DATA_BLOCK DB 5001
VERSION : 0.1
  STRUCT
   MODE_NUM : ARRAY  [0 .. 200 ] OF INT  := 0;
   MODE_LIST_TVS : ARRAY  [1000 .. 1009 ] OF STRUCT
    DINT0 : DINT ;
    DINT1 : DINT ;
    DINT2 : DINT ;
   END_STRUCT ;
   MODE_LIST_TVS1 : ARRAY  [1050 .. 1055 ] OF STRUCT
    DINT0 : DINT ;
    DINT1 : DINT ;
    DINT2 : DINT ;
   END_STRUCT ;
   MODE_LIST_TVS2 : ARRAY  [1130 .. 1135 ] OF STRUCT
    DINT0 : DINT ;
    DINT1 : DINT ;
    DINT2 : DINT ;
   END_STRUCT ;
   MODE_LIST_TVS3 : ARRAY  [1150 .. 1155 ] OF STRUCT
    DINT0 : DINT ;
    DINT1 : DINT ;
    DINT2 : DINT ;
   END_STRUCT ;
   MODE_LIST_TVS4 : ARRAY  [1230 .. 1235 ] OF STRUCT
    DINT0 : DINT ;
    DINT1 : DINT ;
    DINT2 : DINT ;
   END_STRUCT ;
   MODE_LIST_TVS5 : ARRAY  [1250 .. 1255 ] OF STRUCT
    DINT0 : DINT ;
    DINT1 : DINT ;
    DINT2 : DINT ;
   END_STRUCT ;
   MODE_LIST_PVS1 : ARRAY  [2000 .. 2015 ] OF STRUCT
    DINT0 : DINT ;
    DINT1 : DINT ;
    DINT2 : DINT ;
   END_STRUCT ;
   MODE_LIST_PVS2 : ARRAY  [2020 .. 2025 ] OF STRUCT
    DINT0 : DINT ;
    DINT1 : DINT ;
    DINT2 : DINT ;
   END_STRUCT ;
   MODE_LIST_PVS3 : ARRAY  [2050 .. 2065 ] OF STRUCT
    DINT0 : DINT ;
    DINT1 : DINT ;
    DINT2 : DINT ;
   END_STRUCT ;
   MODE_LIST_RVS1 : ARRAY  [3000 .. 3015 ] OF STRUCT
    DINT0 : DINT ;
    DINT1 : DINT ;
    DINT2 : DINT ;
    DINT3 : DINT ;
    DINT4 : DINT ;
    DINT5 : DINT ;
    DINT6 : DINT ;
    DINT7 : DINT ;
    DINT8 : DINT ;
    DINT9 : DINT ;
    DINT10 : DINT ;
   END_STRUCT ;
   MODE_LIST_RVS2 : ARRAY  [3020 .. 3040 ] OF STRUCT
    DINT0 : DINT ;
    DINT1 : DINT ;
    DINT2 : DINT ;
    DINT3 : DINT ;
    DINT4 : DINT ;
    DINT5 : DINT ;
    DINT6 : DINT ;
    DINT7 : DINT ;
    DINT8 : DINT ;
    DINT9 : DINT ;
    DINT10 : DINT ;
   END_STRUCT ;
   MODE_LIST_RVS3 : ARRAY  [3050 .. 3080 ] OF STRUCT
    DINT0 : DINT ;
    DINT1 : DINT ;
    DINT2 : DINT ;
    DINT3 : DINT ;
    DINT4 : DINT ;
    DINT5 : DINT ;
    DINT6 : DINT ;
    DINT7 : DINT ;
    DINT8 : DINT ;
    DINT9 : DINT ;
    DINT10 : DINT ;
   END_STRUCT ;
   MODE_LIST_BY : ARRAY  [3100 .. 3105 ] OF STRUCT
    DINT0 : DINT ;
   END_STRUCT ;
  END_STRUCT ;	
BEGIN
   MODE_NUM[0] := 1000;
   MODE_NUM[1] := 1001;
   MODE_NUM[2] := 1002;
   MODE_NUM[3] := 1003;
   MODE_NUM[4] := 1004;
   MODE_NUM[5] := 1005;
   MODE_NUM[6] := 1006;
   MODE_NUM[7] := 1007;
   MODE_NUM[8] := 1008;
   MODE_NUM[9] := 1009;
   MODE_NUM[10] := 1050;
   MODE_NUM[11] := 1051;
   MODE_NUM[12] := 1052;
   MODE_NUM[13] := 1053;
   MODE_NUM[14] := 1054;
   MODE_NUM[15] := 1055;
   MODE_NUM[16] := 1130;
   MODE_NUM[17] := 1131;
   MODE_NUM[18] := 1132;
   MODE_NUM[19] := 1133;
   MODE_NUM[20] := 1134;
   MODE_NUM[21] := 1135;
   MODE_NUM[22] := 1150;
   MODE_NUM[23] := 1151;
   MODE_NUM[24] := 1152;
   MODE_NUM[25] := 1153;
   MODE_NUM[26] := 1154;
   MODE_NUM[27] := 1155;
   MODE_NUM[28] := 1230;
   MODE_NUM[29] := 1231;
   MODE_NUM[30] := 1232;
   MODE_NUM[31] := 1233;
   MODE_NUM[32] := 1234;
   MODE_NUM[33] := 1235;
   MODE_NUM[34] := 1250;
   MODE_NUM[35] := 1251;
   MODE_NUM[36] := 1252;
   MODE_NUM[37] := 1253;
   MODE_NUM[38] := 1254;
   MODE_NUM[39] := 1255;
   MODE_NUM[40] := 2000;
   MODE_NUM[41] := 2001;
   MODE_NUM[42] := 2002;
   MODE_NUM[43] := 2003;
   MODE_NUM[44] := 2004;
   MODE_NUM[45] := 2005;
   MODE_NUM[46] := 2006;
   MODE_NUM[47] := 2007;
   MODE_NUM[48] := 2008;
   MODE_NUM[49] := 2009;
   MODE_NUM[50] := 2010;
   MODE_NUM[51] := 2011;
   MODE_NUM[52] := 2012;
   MODE_NUM[53] := 2013;
   MODE_NUM[54] := 2014;
   MODE_NUM[55] := 2015;
   MODE_NUM[56] := 2020;
   MODE_NUM[57] := 2021;
   MODE_NUM[58] := 2022;
   MODE_NUM[59] := 2023;
   MODE_NUM[60] := 2024;
   MODE_NUM[61] := 2025;
   MODE_NUM[62] := 2050;
   MODE_NUM[63] := 2051;
   MODE_NUM[64] := 2052;
   MODE_NUM[65] := 2053;
   MODE_NUM[66] := 2054;
   MODE_NUM[67] := 2055;
   MODE_NUM[68] := 2056;
   MODE_NUM[69] := 2057;
   MODE_NUM[70] := 2058;
   MODE_NUM[71] := 2059;
   MODE_NUM[72] := 2060;
   MODE_NUM[73] := 2061;
   MODE_NUM[74] := 2062;
   MODE_NUM[75] := 2063;
   MODE_NUM[76] := 2064;
   MODE_NUM[77] := 2065;
   MODE_NUM[78] := 3000;
   MODE_NUM[79] := 3001;
   MODE_NUM[80] := 3002;
   MODE_NUM[81] := 3003;
   MODE_NUM[82] := 3004;
   MODE_NUM[83] := 3005;
   MODE_NUM[84] := 3006;
   MODE_NUM[85] := 3007;
   MODE_NUM[86] := 3008;
   MODE_NUM[87] := 3009;
   MODE_NUM[88] := 3010;
   MODE_NUM[89] := 302;
   MODE_NUM[90] := 3012;
   MODE_NUM[91] := 3013;
   MODE_NUM[92] := 3014;
   MODE_NUM[93] := 3015;
   MODE_NUM[94] := 3020;
   MODE_NUM[95] := 3021;
   MODE_NUM[96] := 3022;
   MODE_NUM[97] := 3023;
   MODE_NUM[98] := 3024;
   MODE_NUM[99] := 3025;
   MODE_NUM[100] := 3026;
   MODE_NUM[101] := 3027;
   MODE_NUM[102] := 3028;
   MODE_NUM[103] := 3029;
   MODE_NUM[104] := 3030;
   MODE_NUM[105] := 3031;
   MODE_NUM[106] := 3032;
   MODE_NUM[107] := 3033;
   MODE_NUM[108] := 3034;
   MODE_NUM[109] := 3035;
   MODE_NUM[110] := 3036;
   MODE_NUM[111] := 3037;
   MODE_NUM[112] := 3038;
   MODE_NUM[113] := 3039;
   MODE_NUM[114] := 3040;
   MODE_NUM[115] := 3050;
   MODE_NUM[116] := 3051;
   MODE_NUM[117] := 3052;
   MODE_NUM[118] := 3053;
   MODE_NUM[119] := 3054;
   MODE_NUM[120] := 3055;
   MODE_NUM[121] := 3056;
   MODE_NUM[122] := 3057;
   MODE_NUM[123] := 3058;
   MODE_NUM[124] := 3059;
   MODE_NUM[125] := 3060;
   MODE_NUM[126] := 3061;
   MODE_NUM[127] := 3062;
   MODE_NUM[128] := 3063;
   MODE_NUM[129] := 3064;
   MODE_NUM[130] := 3065;
   MODE_NUM[131] := 3066;
   MODE_NUM[132] := 3067;
   MODE_NUM[133] := 3068;
   MODE_NUM[134] := 3069;
   MODE_NUM[135] := 3070;
   MODE_NUM[136] := 3071;
   MODE_NUM[137] := 3072;
   MODE_NUM[138] := 3073;
   MODE_NUM[139] := 3074;
   MODE_NUM[140] := 3075;
   MODE_NUM[141] := 3076;
   MODE_NUM[142] := 3077;
   MODE_NUM[143] := 3078;
   MODE_NUM[144] := 3079;
   MODE_NUM[145] := 3080;
   MODE_LIST_TVS[1000].DINT0 := L#1475696127;
   MODE_LIST_TVS[1000].DINT1 := L#1431697397;
   MODE_LIST_TVS[1001].DINT0 := L#-580919467;
   MODE_LIST_TVS[1001].DINT1 := L#-8865;
   MODE_LIST_TVS[1002].DINT0 := L#-44171350;
   MODE_LIST_TVS[1002].DINT1 := L#-33443;
   MODE_LIST_TVS[1003].DINT0 := L#-547496107;
   MODE_LIST_TVS[1003].DINT1 := L#1431699293;
   MODE_LIST_TVS[1004].DINT0 := L#-547496022;
   MODE_LIST_TVS[1004].DINT1 := L#1431699293;
   MODE_LIST_TVS[1005].DINT0 := L#1609916415;
   MODE_LIST_TVS[1005].DINT1 := L#1431699445;
   MODE_LIST_TVS1[1050].DINT0 := L#-142779785;
   MODE_LIST_TVS1[1050].DINT1 := L#-572655747;
   MODE_LIST_TVS1[1051].DINT0 := L#-673850659;
   MODE_LIST_TVS1[1051].DINT1 := L#-572655649;
   MODE_LIST_TVS1[1052].DINT0 := L#-142779785;
   MODE_LIST_TVS1[1052].DINT1 := L#-572688513;
   MODE_LIST_TVS1[1053].DINT0 := L#-136979747;
   MODE_LIST_TVS1[1053].DINT1 := L#-572663841;
   MODE_LIST_TVS4[1230].DINT0 := L#1609916351;
   MODE_LIST_TVS4[1230].DINT1 := L#1431699325;
   MODE_LIST_TVS4[1231].DINT0 := L#-537567249;
   MODE_LIST_TVS4[1231].DINT1 := L#1431699413;
   MODE_LIST_TVS4[1232].DINT0 := L#-537567313;
   MODE_LIST_TVS4[1232].DINT1 := L#1431699293;
   MODE_LIST_TVS5[1250].DINT0 := L#-142779817;
   MODE_LIST_TVS5[1250].DINT1 := L#-572656291;
   MODE_LIST_TVS5[1251].DINT0 := L#1602052027;
   MODE_LIST_TVS5[1251].DINT1 := L#1431699325;
   MODE_LIST_TVS5[1252].DINT0 := L#-539631634;
   MODE_LIST_TVS5[1252].DINT1 := L#1431699413;
   MODE_LIST_TVS5[1253].DINT0 := L#-673850787;
   MODE_LIST_TVS5[1253].DINT1 := L#-572656289;
   MODE_LIST_PVS1[2000].DINT0 := L#-356515841;
   MODE_LIST_PVS1[2000].DINT1 := L#-1;
   MODE_LIST_PVS1[2000].DINT2 := L#16383;
   MODE_LIST_PVS1[2001].DINT0 := L#-356518571;
   MODE_LIST_PVS1[2001].DINT1 := L#-305291;
   MODE_LIST_PVS1[2001].DINT2 := L#15735;
   MODE_LIST_PVS1[2002].DINT0 := L#1790965077;
   MODE_LIST_PVS1[2002].DINT1 := L#-41515;
   MODE_LIST_PVS1[2002].DINT2 := L#15829;
   MODE_LIST_PVS1[2003].DINT0 := L#1790965077;
   MODE_LIST_PVS1[2003].DINT1 := L#-41515;
   MODE_LIST_PVS1[2003].DINT2 := L#15829;
   MODE_LIST_PVS1[2004].DINT0 := L#1790965077;
   MODE_LIST_PVS1[2004].DINT1 := L#-41515;
   MODE_LIST_PVS1[2004].DINT2 := L#15829;
   MODE_LIST_PVS1[2005].DINT0 := L#-1;
   MODE_LIST_PVS1[2005].DINT1 := L#-1;
   MODE_LIST_PVS1[2005].DINT2 := L#16383;
   MODE_LIST_PVS1[2006].DINT0 := L#1434449237;
   MODE_LIST_PVS1[2006].DINT1 := L#3888469;
   MODE_LIST_PVS1[2006].DINT2 := L#15701;
   MODE_LIST_PVS1[2007].DINT0 := L#1790967765;
   MODE_LIST_PVS1[2007].DINT1 := L#4194293;
   MODE_LIST_PVS1[2007].DINT2 := L#16373;
   MODE_LIST_PVS1[2008].DINT0 := L#-356518529;
   MODE_LIST_PVS1[2008].DINT1 := L#4152799;
   MODE_LIST_PVS1[2008].DINT2 := L#15839;
   MODE_LIST_PVS1[2009].DINT0 := L#-1;
   MODE_LIST_PVS1[2009].DINT1 := L#-1;
   MODE_LIST_PVS1[2009].DINT2 := L#16383;
   MODE_LIST_PVS1[2010].DINT0 := L#-143261697;
   MODE_LIST_PVS1[2010].DINT1 := L#4059103;
   MODE_LIST_PVS1[2010].DINT2 := L#14335;
   MODE_LIST_PVS1[2011].DINT0 := L#-143261697;
   MODE_LIST_PVS1[2011].DINT1 := L#4059103;
   MODE_LIST_PVS1[2011].DINT2 := L#14335;
   MODE_LIST_PVS3[2050].DINT0 := L#-1019224065;
   MODE_LIST_PVS3[2050].DINT1 := L#3670015;
   MODE_LIST_PVS3[2050].DINT2 := L#16383;
   MODE_LIST_PVS3[2051].DINT0 := L#-600309761;
   MODE_LIST_PVS3[2051].DINT1 := L#4194303;
   MODE_LIST_PVS3[2051].DINT2 := L#14335;
   MODE_LIST_PVS3[2052].DINT0 := L#-1069580289;
   MODE_LIST_PVS3[2052].DINT1 := L#2145386495;
   MODE_LIST_PVS3[2052].DINT2 := L#16383;
   MODE_LIST_PVS3[2053].DINT0 := L#-1069580289;
   MODE_LIST_PVS3[2053].DINT1 := L#-10485761;
   MODE_LIST_PVS3[2053].DINT2 := L#16383;
   MODE_LIST_PVS3[2054].DINT0 := L#-1069580289;
   MODE_LIST_PVS3[2054].DINT1 := L#-673185793;
   MODE_LIST_PVS3[2054].DINT2 := L#16383;
   MODE_LIST_PVS3[2055].DINT0 := L#-1069580289;
   MODE_LIST_PVS3[2055].DINT1 := L#-35651585;
   MODE_LIST_PVS3[2055].DINT2 := L#16383;
   MODE_LIST_PVS3[2056].DINT0 := L#-1071644673;
   MODE_LIST_PVS3[2056].DINT1 := L#4194303;
   MODE_LIST_PVS3[2056].DINT2 := L#8191;
   MODE_LIST_PVS3[2057].DINT0 := L#-143261697;
   MODE_LIST_PVS3[2057].DINT1 := L#4059103;
   MODE_LIST_PVS3[2057].DINT2 := L#14335;
   MODE_LIST_RVS1[3000].DINT0 := L#1431666687;
   MODE_LIST_RVS1[3000].DINT1 := L#-11;
   MODE_LIST_RVS1[3000].DINT2 := L#-1;
   MODE_LIST_RVS1[3000].DINT3 := L#1431656447;
   MODE_LIST_RVS1[3000].DINT4 := L#1431655765;
   MODE_LIST_RVS1[3000].DINT5 := L#-43;
   MODE_LIST_RVS1[3000].DINT6 := L#-1;
   MODE_LIST_RVS1[3000].DINT7 := L#1432354815;
   MODE_LIST_RVS1[3000].DINT8 := L#-43691;
   MODE_LIST_RVS1[3000].DINT9 := L#-1;
   MODE_LIST_RVS1[3000].DINT10 := L#255;
   MODE_LIST_RVS1[3001].DINT0 := L#16383;
   MODE_LIST_RVS1[3001].DINT1 := L#-16;
   MODE_LIST_RVS1[3001].DINT2 := L#-1;
   MODE_LIST_RVS1[3001].DINT3 := L#1023;
   MODE_LIST_RVS1[3001].DINT5 := L#-64;
   MODE_LIST_RVS1[3001].DINT6 := L#-1;
   MODE_LIST_RVS1[3001].DINT7 := L#1048575;
   MODE_LIST_RVS1[3001].DINT8 := L#-65536;
   MODE_LIST_RVS1[3001].DINT9 := L#-1;
   MODE_LIST_RVS1[3001].DINT10 := L#255;
   MODE_LIST_RVS1[3002].DINT0 := L#10069;
   MODE_LIST_RVS1[3002].DINT1 := L#-707406000;
   MODE_LIST_RVS1[3002].DINT2 := L#1507164117;
   MODE_LIST_RVS1[3002].DINT3 := L#629;
   MODE_LIST_RVS1[3002].DINT5 := L#2012599616;
   MODE_LIST_RVS1[3002].DINT6 := L#-170568363;
   MODE_LIST_RVS1[3002].DINT7 := L#644479;
   MODE_LIST_RVS1[3002].DINT8 := L#1567948800;
   MODE_LIST_RVS1[3002].DINT9 := L#1567972725;
   MODE_LIST_RVS1[3002].DINT10 := L#255;
   MODE_LIST_RVS1[3003].DINT0 := L#7509;
   MODE_LIST_RVS1[3003].DINT1 := L#-707406000;
   MODE_LIST_RVS1[3003].DINT2 := L#1465221077;
   MODE_LIST_RVS1[3003].DINT3 := L#469;
   MODE_LIST_RVS1[3003].DINT5 := L#2012599616;
   MODE_LIST_RVS1[3003].DINT6 := L#-170568363;
   MODE_LIST_RVS1[3003].DINT7 := L#480639;
   MODE_LIST_RVS1[3003].DINT8 := L#1567948800;
   MODE_LIST_RVS1[3003].DINT9 := L#1567972725;
   MODE_LIST_RVS1[3003].DINT10 := L#255;
   MODE_LIST_RVS1[3004].DINT0 := L#7509;
   MODE_LIST_RVS1[3004].DINT1 := L#-707406000;
   MODE_LIST_RVS1[3004].DINT2 := L#1465221077;
   MODE_LIST_RVS1[3004].DINT3 := L#469;
   MODE_LIST_RVS1[3004].DINT5 := L#1442174272;
   MODE_LIST_RVS1[3004].DINT6 := L#-170568363;
   MODE_LIST_RVS1[3004].DINT7 := L#480639;
   MODE_LIST_RVS1[3004].DINT8 := L#1567948800;
   MODE_LIST_RVS1[3004].DINT9 := L#1567972725;
   MODE_LIST_RVS1[3004].DINT10 := L#255;
   MODE_LIST_RVS1[3005].DINT0 := L#7509;
   MODE_LIST_RVS1[3005].DINT1 := L#-707406000;
   MODE_LIST_RVS1[3005].DINT2 := L#1507164117;
   MODE_LIST_RVS1[3005].DINT3 := L#469;
   MODE_LIST_RVS1[3005].DINT5 := L#1442174272;
   MODE_LIST_RVS1[3005].DINT6 := L#-170568363;
   MODE_LIST_RVS1[3005].DINT7 := L#480639;
   MODE_LIST_RVS1[3005].DINT8 := L#1567948800;
   MODE_LIST_RVS1[3005].DINT9 := L#1567972725;
   MODE_LIST_RVS1[3005].DINT10 := L#255;
   MODE_LIST_RVS1[3006].DINT0 := L#16383;
   MODE_LIST_RVS1[3006].DINT1 := L#-16;
   MODE_LIST_RVS1[3006].DINT2 := L#-10944;
   MODE_LIST_RVS1[3006].DINT3 := L#1023;
   MODE_LIST_RVS1[3006].DINT5 := L#-8521792;
   MODE_LIST_RVS1[3006].DINT6 := L#2147221504;
   MODE_LIST_RVS1[3006].DINT7 := L#1048533;
   MODE_LIST_RVS1[3006].DINT8 := L#268369920;
   MODE_LIST_RVS1[3006].DINT9 := L#268374015;
   MODE_LIST_RVS1[3006].DINT10 := L#85;
   MODE_LIST_RVS2[3020].DINT0 := L#1431657813;
   MODE_LIST_RVS2[3020].DINT1 := L#-11;
   MODE_LIST_RVS2[3020].DINT2 := L#-64;
   MODE_LIST_RVS2[3020].DINT3 := L#1023;
   MODE_LIST_RVS2[3020].DINT5 := L#-8521792;
   MODE_LIST_RVS2[3020].DINT6 := L#-262144;
   MODE_LIST_RVS2[3020].DINT7 := L#1048575;
   MODE_LIST_RVS2[3020].DINT8 := L#268369920;
   MODE_LIST_RVS2[3020].DINT9 := L#268374015;
   MODE_LIST_RVS2[3020].DINT10 := L#255;
   MODE_LIST_RVS2[3021].DINT0 := L#1431657813;
   MODE_LIST_RVS2[3021].DINT1 := L#-11;
   MODE_LIST_RVS2[3021].DINT2 := L#-64;
   MODE_LIST_RVS2[3021].DINT3 := L#1023;
   MODE_LIST_RVS2[3021].DINT5 := L#-8521792;
   MODE_LIST_RVS2[3021].DINT6 := L#-262144;
   MODE_LIST_RVS2[3021].DINT7 := L#1048575;
   MODE_LIST_RVS2[3021].DINT8 := L#268369920;
   MODE_LIST_RVS2[3021].DINT9 := L#268374015;
   MODE_LIST_RVS2[3021].DINT10 := L#255;
   MODE_LIST_RVS2[3022].DINT0 := L#1431657813;
   MODE_LIST_RVS2[3022].DINT1 := L#-11;
   MODE_LIST_RVS2[3022].DINT2 := L#-64;
   MODE_LIST_RVS2[3022].DINT3 := L#1023;
   MODE_LIST_RVS2[3022].DINT5 := L#-8521792;
   MODE_LIST_RVS2[3022].DINT6 := L#-262144;
   MODE_LIST_RVS2[3022].DINT7 := L#1048575;
   MODE_LIST_RVS2[3022].DINT8 := L#268369920;
   MODE_LIST_RVS2[3022].DINT9 := L#268374015;
   MODE_LIST_RVS2[3022].DINT10 := L#255;
   MODE_LIST_RVS2[3023].DINT0 := L#1431657813;
   MODE_LIST_RVS2[3023].DINT1 := L#-11;
   MODE_LIST_RVS2[3023].DINT2 := L#-64;
   MODE_LIST_RVS2[3023].DINT3 := L#1023;
   MODE_LIST_RVS2[3023].DINT5 := L#-8521792;
   MODE_LIST_RVS2[3023].DINT6 := L#-262144;
   MODE_LIST_RVS2[3023].DINT7 := L#1048575;
   MODE_LIST_RVS2[3023].DINT8 := L#268369920;
   MODE_LIST_RVS2[3023].DINT9 := L#268374015;
   MODE_LIST_RVS2[3023].DINT10 := L#255;
   MODE_LIST_RVS2[3024].DINT0 := L#16383;
   MODE_LIST_RVS2[3024].DINT1 := L#-16;
   MODE_LIST_RVS2[3024].DINT2 := L#1610612672;
   MODE_LIST_RVS2[3024].DINT3 := L#1431655893;
   MODE_LIST_RVS2[3024].DINT4 := L#1431655765;
   MODE_LIST_RVS2[3024].DINT5 := L#-8521771;
   MODE_LIST_RVS2[3024].DINT6 := L#-262144;
   MODE_LIST_RVS2[3024].DINT7 := L#1048575;
   MODE_LIST_RVS2[3024].DINT8 := L#268369920;
   MODE_LIST_RVS2[3024].DINT9 := L#268374015;
   MODE_LIST_RVS2[3024].DINT10 := L#255;
   MODE_LIST_RVS2[3025].DINT0 := L#16383;
   MODE_LIST_RVS2[3025].DINT1 := L#-16;
   MODE_LIST_RVS2[3025].DINT2 := L#1610612672;
   MODE_LIST_RVS2[3025].DINT3 := L#1431655893;
   MODE_LIST_RVS2[3025].DINT4 := L#1431655765;
   MODE_LIST_RVS2[3025].DINT5 := L#-8521771;
   MODE_LIST_RVS2[3025].DINT6 := L#-262144;
   MODE_LIST_RVS2[3025].DINT7 := L#1048575;
   MODE_LIST_RVS2[3025].DINT8 := L#268369920;
   MODE_LIST_RVS2[3025].DINT9 := L#268374015;
   MODE_LIST_RVS2[3025].DINT10 := L#255;
   MODE_LIST_RVS2[3026].DINT0 := L#16383;
   MODE_LIST_RVS2[3026].DINT1 := L#-16;
   MODE_LIST_RVS2[3026].DINT2 := L#1610612672;
   MODE_LIST_RVS2[3026].DINT3 := L#1431655893;
   MODE_LIST_RVS2[3026].DINT4 := L#1431655765;
   MODE_LIST_RVS2[3026].DINT5 := L#-8521771;
   MODE_LIST_RVS2[3026].DINT6 := L#-262144;
   MODE_LIST_RVS2[3026].DINT7 := L#1048575;
   MODE_LIST_RVS2[3026].DINT8 := L#268369920;
   MODE_LIST_RVS2[3026].DINT9 := L#268374015;
   MODE_LIST_RVS2[3026].DINT10 := L#255;
   MODE_LIST_RVS2[3027].DINT0 := L#16383;
   MODE_LIST_RVS2[3027].DINT1 := L#-16;
   MODE_LIST_RVS2[3027].DINT2 := L#1610612672;
   MODE_LIST_RVS2[3027].DINT3 := L#1431655893;
   MODE_LIST_RVS2[3027].DINT4 := L#1431655765;
   MODE_LIST_RVS2[3027].DINT5 := L#-8521771;
   MODE_LIST_RVS2[3027].DINT6 := L#-262144;
   MODE_LIST_RVS2[3027].DINT7 := L#1048575;
   MODE_LIST_RVS2[3027].DINT8 := L#268369920;
   MODE_LIST_RVS2[3027].DINT9 := L#268374015;
   MODE_LIST_RVS2[3027].DINT10 := L#255;
   MODE_LIST_RVS2[3028].DINT0 := L#16383;
   MODE_LIST_RVS2[3028].DINT1 := L#-16;
   MODE_LIST_RVS2[3028].DINT2 := L#1610612672;
   MODE_LIST_RVS2[3028].DINT3 := L#1431655893;
   MODE_LIST_RVS2[3028].DINT4 := L#1431655765;
   MODE_LIST_RVS2[3028].DINT5 := L#-8521771;
   MODE_LIST_RVS2[3028].DINT6 := L#-262144;
   MODE_LIST_RVS2[3028].DINT7 := L#1048575;
   MODE_LIST_RVS2[3028].DINT8 := L#268369920;
   MODE_LIST_RVS2[3028].DINT9 := L#268374015;
   MODE_LIST_RVS2[3028].DINT10 := L#255;
   MODE_LIST_RVS2[3029].DINT0 := L#16383;
   MODE_LIST_RVS2[3029].DINT1 := L#-16;
   MODE_LIST_RVS2[3029].DINT2 := L#1610612672;
   MODE_LIST_RVS2[3029].DINT3 := L#1431655893;
   MODE_LIST_RVS2[3029].DINT4 := L#1431655765;
   MODE_LIST_RVS2[3029].DINT5 := L#-8521771;
   MODE_LIST_RVS2[3029].DINT6 := L#-262144;
   MODE_LIST_RVS2[3029].DINT7 := L#1048575;
   MODE_LIST_RVS2[3029].DINT8 := L#268369920;
   MODE_LIST_RVS2[3029].DINT9 := L#268374015;
   MODE_LIST_RVS2[3029].DINT10 := L#255;
   MODE_LIST_RVS2[3030].DINT0 := L#16383;
   MODE_LIST_RVS2[3030].DINT1 := L#-16;
   MODE_LIST_RVS2[3030].DINT2 := L#1610612672;
   MODE_LIST_RVS2[3030].DINT3 := L#1431655893;
   MODE_LIST_RVS2[3030].DINT4 := L#1431655765;
   MODE_LIST_RVS2[3030].DINT5 := L#-8521771;
   MODE_LIST_RVS2[3030].DINT6 := L#-262144;
   MODE_LIST_RVS2[3030].DINT7 := L#1048575;
   MODE_LIST_RVS2[3030].DINT8 := L#268369920;
   MODE_LIST_RVS2[3030].DINT9 := L#268374015;
   MODE_LIST_RVS2[3030].DINT10 := L#255;
   MODE_LIST_RVS2[3031].DINT0 := L#16383;
   MODE_LIST_RVS2[3031].DINT1 := L#-16;
   MODE_LIST_RVS2[3031].DINT2 := L#1610612672;
   MODE_LIST_RVS2[3031].DINT3 := L#1431655893;
   MODE_LIST_RVS2[3031].DINT4 := L#1431655765;
   MODE_LIST_RVS2[3031].DINT5 := L#-8521771;
   MODE_LIST_RVS2[3031].DINT6 := L#-262144;
   MODE_LIST_RVS2[3031].DINT7 := L#1048575;
   MODE_LIST_RVS2[3031].DINT8 := L#268369920;
   MODE_LIST_RVS2[3031].DINT9 := L#268374015;
   MODE_LIST_RVS2[3031].DINT10 := L#255;
   MODE_LIST_RVS2[3032].DINT0 := L#16383;
   MODE_LIST_RVS2[3032].DINT1 := L#-16;
   MODE_LIST_RVS2[3032].DINT2 := L#1610612672;
   MODE_LIST_RVS2[3032].DINT3 := L#1431655893;
   MODE_LIST_RVS2[3032].DINT4 := L#1431655765;
   MODE_LIST_RVS2[3032].DINT5 := L#-8521771;
   MODE_LIST_RVS2[3032].DINT6 := L#-262144;
   MODE_LIST_RVS2[3032].DINT7 := L#1048575;
   MODE_LIST_RVS2[3032].DINT8 := L#268369920;
   MODE_LIST_RVS2[3032].DINT9 := L#268374015;
   MODE_LIST_RVS2[3032].DINT10 := L#255;
   MODE_LIST_RVS2[3033].DINT0 := L#16383;
   MODE_LIST_RVS2[3033].DINT1 := L#-16;
   MODE_LIST_RVS2[3033].DINT2 := L#1610612672;
   MODE_LIST_RVS2[3033].DINT3 := L#1431655893;
   MODE_LIST_RVS2[3033].DINT4 := L#1431655765;
   MODE_LIST_RVS2[3033].DINT5 := L#-8521771;
   MODE_LIST_RVS2[3033].DINT6 := L#-262144;
   MODE_LIST_RVS2[3033].DINT7 := L#1048575;
   MODE_LIST_RVS2[3033].DINT8 := L#268369920;
   MODE_LIST_RVS2[3033].DINT9 := L#268374015;
   MODE_LIST_RVS2[3033].DINT10 := L#255;
   MODE_LIST_RVS2[3034].DINT0 := L#4178175;
   MODE_LIST_RVS2[3034].DINT2 := L#65280;
   MODE_LIST_RVS2[3034].DINT3 := L#1073725440;
   MODE_LIST_RVS2[3034].DINT5 := L#-8521792;
   MODE_LIST_RVS2[3034].DINT6 := L#-262144;
   MODE_LIST_RVS2[3034].DINT7 := L#-16777153;
   MODE_LIST_RVS2[3034].DINT8 := L#-66060289;
   MODE_LIST_RVS2[3034].DINT9 := L#1073741823;
   MODE_LIST_RVS2[3035].DINT0 := L#16383;
   MODE_LIST_RVS2[3035].DINT1 := L#-16;
   MODE_LIST_RVS2[3035].DINT2 := L#-64;
   MODE_LIST_RVS2[3035].DINT3 := L#1023;
   MODE_LIST_RVS2[3035].DINT5 := L#-8521792;
   MODE_LIST_RVS2[3035].DINT6 := L#-262144;
   MODE_LIST_RVS2[3035].DINT7 := L#1431786879;
   MODE_LIST_RVS2[3035].DINT8 := L#268391765;
   MODE_LIST_RVS2[3035].DINT9 := L#268374015;
   MODE_LIST_RVS2[3035].DINT10 := L#255;
   MODE_LIST_RVS2[3036].DINT0 := L#16383;
   MODE_LIST_RVS2[3036].DINT1 := L#-16;
   MODE_LIST_RVS2[3036].DINT2 := L#-64;
   MODE_LIST_RVS2[3036].DINT3 := L#1023;
   MODE_LIST_RVS2[3036].DINT5 := L#-8521792;
   MODE_LIST_RVS2[3036].DINT6 := L#-262144;
   MODE_LIST_RVS2[3036].DINT7 := L#1431786879;
   MODE_LIST_RVS2[3036].DINT8 := L#268391765;
   MODE_LIST_RVS2[3036].DINT9 := L#268374015;
   MODE_LIST_RVS2[3036].DINT10 := L#255;
   MODE_LIST_RVS2[3037].DINT0 := L#16383;
   MODE_LIST_RVS2[3037].DINT1 := L#-16;
   MODE_LIST_RVS2[3037].DINT2 := L#-64;
   MODE_LIST_RVS2[3037].DINT3 := L#1023;
   MODE_LIST_RVS2[3037].DINT5 := L#-8521792;
   MODE_LIST_RVS2[3037].DINT6 := L#-262144;
   MODE_LIST_RVS2[3037].DINT7 := L#1431786879;
   MODE_LIST_RVS2[3037].DINT8 := L#268391765;
   MODE_LIST_RVS2[3037].DINT9 := L#268374015;
   MODE_LIST_RVS2[3037].DINT10 := L#255;
   MODE_LIST_RVS2[3038].DINT0 := L#16383;
   MODE_LIST_RVS2[3038].DINT1 := L#-16;
   MODE_LIST_RVS2[3038].DINT2 := L#-64;
   MODE_LIST_RVS2[3038].DINT3 := L#1023;
   MODE_LIST_RVS2[3038].DINT5 := L#-8521792;
   MODE_LIST_RVS2[3038].DINT6 := L#-262144;
   MODE_LIST_RVS2[3038].DINT7 := L#1431786879;
   MODE_LIST_RVS2[3038].DINT8 := L#268391765;
   MODE_LIST_RVS2[3038].DINT9 := L#268374015;
   MODE_LIST_RVS2[3038].DINT10 := L#255;
   MODE_LIST_RVS2[3039].DINT0 := L#16383;
   MODE_LIST_RVS2[3039].DINT1 := L#-16;
   MODE_LIST_RVS2[3039].DINT2 := L#-64;
   MODE_LIST_RVS2[3039].DINT3 := L#1023;
   MODE_LIST_RVS2[3039].DINT5 := L#-8521792;
   MODE_LIST_RVS2[3039].DINT6 := L#-262144;
   MODE_LIST_RVS2[3039].DINT7 := L#1431786879;
   MODE_LIST_RVS2[3039].DINT8 := L#268391765;
   MODE_LIST_RVS2[3039].DINT9 := L#268374015;
   MODE_LIST_RVS2[3039].DINT10 := L#255;
   MODE_LIST_RVS3[3050].DINT0 := L#-1;
   MODE_LIST_RVS3[3050].DINT1 := L#255;
   MODE_LIST_RVS3[3050].DINT2 := L#4194048;
   MODE_LIST_RVS3[3050].DINT3 := L#-581091328;
   MODE_LIST_RVS3[3050].DINT4 := L#262133;
   MODE_LIST_RVS3[3050].DINT5 := L#-8521792;
   MODE_LIST_RVS3[3050].DINT6 := L#2147221504;
   MODE_LIST_RVS3[3050].DINT7 := L#1007681493;
   MODE_LIST_RVS3[3050].DINT8 := L#-168296512;
   MODE_LIST_RVS3[3050].DINT9 := L#-43523;
   MODE_LIST_RVS3[3050].DINT10 := L#4095;
   MODE_LIST_RVS3[3051].DINT0 := L#268435455;
   MODE_LIST_RVS3[3051].DINT1 := L#15;
   MODE_LIST_RVS3[3051].DINT2 := L#4194048;
   MODE_LIST_RVS3[3051].DINT3 := L#-581091328;
   MODE_LIST_RVS3[3051].DINT4 := L#262133;
   MODE_LIST_RVS3[3051].DINT5 := L#-8521792;
   MODE_LIST_RVS3[3051].DINT6 := L#2147221504;
   MODE_LIST_RVS3[3051].DINT7 := L#-1070530603;
   MODE_LIST_RVS3[3051].DINT8 := L#-168296512;
   MODE_LIST_RVS3[3051].DINT9 := L#-43523;
   MODE_LIST_RVS3[3051].DINT10 := L#4095;
   MODE_LIST_RVS3[3052].DINT0 := L#12599295;
   MODE_LIST_RVS3[3052].DINT1 := L#-4;
   MODE_LIST_RVS3[3052].DINT2 := L#-10944;
   MODE_LIST_RVS3[3052].DINT3 := L#1023;
   MODE_LIST_RVS3[3052].DINT5 := L#-8521792;
   MODE_LIST_RVS3[3052].DINT6 := L#2147221504;
   MODE_LIST_RVS3[3052].DINT7 := L#1048533;
   MODE_LIST_RVS3[3052].DINT8 := L#268369920;
   MODE_LIST_RVS3[3052].DINT9 := L#268374015;
   MODE_LIST_RVS3[3052].DINT10 := L#85;
   MODE_LIST_RVS3[3053].DINT0 := L#-1070579713;
   MODE_LIST_RVS3[3053].DINT1 := L#-13;
   MODE_LIST_RVS3[3053].DINT2 := L#-10944;
   MODE_LIST_RVS3[3053].DINT3 := L#1023;
   MODE_LIST_RVS3[3053].DINT5 := L#-8521792;
   MODE_LIST_RVS3[3053].DINT6 := L#2147221504;
   MODE_LIST_RVS3[3053].DINT7 := L#1048533;
   MODE_LIST_RVS3[3053].DINT8 := L#268369920;
   MODE_LIST_RVS3[3053].DINT9 := L#268374015;
   MODE_LIST_RVS3[3053].DINT10 := L#85;
   MODE_LIST_RVS3[3054].DINT0 := L#16383;
   MODE_LIST_RVS3[3054].DINT1 := L#-16;
   MODE_LIST_RVS3[3054].DINT2 := L#-10944;
   MODE_LIST_RVS3[3054].DINT3 := L#1023;
   MODE_LIST_RVS3[3054].DINT5 := L#-8521792;
   MODE_LIST_RVS3[3054].DINT6 := L#2147221504;
   MODE_LIST_RVS3[3054].DINT7 := L#1048533;
   MODE_LIST_RVS3[3054].DINT8 := L#268369920;
   MODE_LIST_RVS3[3054].DINT9 := L#268374015;
   MODE_LIST_RVS3[3054].DINT10 := L#85;
   MODE_LIST_RVS3[3055].DINT0 := L#16383;
   MODE_LIST_RVS3[3055].DINT1 := L#-35376;
   MODE_LIST_RVS3[3055].DINT2 := L#-10944;
   MODE_LIST_RVS3[3055].DINT3 := L#1023;
   MODE_LIST_RVS3[3055].DINT5 := L#-8521792;
   MODE_LIST_RVS3[3055].DINT6 := L#2147221504;
   MODE_LIST_RVS3[3055].DINT7 := L#1048533;
   MODE_LIST_RVS3[3055].DINT8 := L#268369920;
   MODE_LIST_RVS3[3055].DINT9 := L#268374015;
   MODE_LIST_RVS3[3055].DINT10 := L#85;
   MODE_LIST_RVS3[3056].DINT0 := L#16383;
   MODE_LIST_RVS3[3056].DINT1 := L#2105409520;
   MODE_LIST_RVS3[3056].DINT2 := L#-10881;
   MODE_LIST_RVS3[3056].DINT3 := L#1023;
   MODE_LIST_RVS3[3056].DINT5 := L#-8521792;
   MODE_LIST_RVS3[3056].DINT6 := L#2147221504;
   MODE_LIST_RVS3[3056].DINT7 := L#1048533;
   MODE_LIST_RVS3[3056].DINT8 := L#268369920;
   MODE_LIST_RVS3[3056].DINT9 := L#268374015;
   MODE_LIST_RVS3[3056].DINT10 := L#85;
   MODE_LIST_RVS3[3057].DINT0 := L#16383;
   MODE_LIST_RVS3[3057].DINT1 := L#-16;
   MODE_LIST_RVS3[3057].DINT2 := L#-10944;
   MODE_LIST_RVS3[3057].DINT3 := L#1023;
   MODE_LIST_RVS3[3057].DINT5 := L#-8521792;
   MODE_LIST_RVS3[3057].DINT6 := L#2147221504;
   MODE_LIST_RVS3[3057].DINT7 := L#1048533;
   MODE_LIST_RVS3[3057].DINT8 := L#268369920;
   MODE_LIST_RVS3[3057].DINT9 := L#268374015;
   MODE_LIST_RVS3[3057].DINT10 := L#85;
   MODE_LIST_RVS3[3058].DINT0 := L#16383;
   MODE_LIST_RVS3[3058].DINT1 := L#-16;
   MODE_LIST_RVS3[3058].DINT2 := L#-10944;
   MODE_LIST_RVS3[3058].DINT3 := L#201327615;
   MODE_LIST_RVS3[3058].DINT4 := L#50331648;
   MODE_LIST_RVS3[3058].DINT5 := L#-8521792;
   MODE_LIST_RVS3[3058].DINT6 := L#2147221504;
   MODE_LIST_RVS3[3058].DINT7 := L#1048533;
   MODE_LIST_RVS3[3058].DINT8 := L#268369920;
   MODE_LIST_RVS3[3058].DINT9 := L#268374015;
   MODE_LIST_RVS3[3058].DINT10 := L#85;
   MODE_LIST_RVS3[3059].DINT0 := L#16383;
   MODE_LIST_RVS3[3059].DINT1 := L#-16;
   MODE_LIST_RVS3[3059].DINT2 := L#-10944;
   MODE_LIST_RVS3[3059].DINT3 := L#805307391;
   MODE_LIST_RVS3[3059].DINT4 := L#201326592;
   MODE_LIST_RVS3[3059].DINT5 := L#-8521792;
   MODE_LIST_RVS3[3059].DINT6 := L#2147221504;
   MODE_LIST_RVS3[3059].DINT7 := L#1048533;
   MODE_LIST_RVS3[3059].DINT8 := L#268369920;
   MODE_LIST_RVS3[3059].DINT9 := L#268374015;
   MODE_LIST_RVS3[3059].DINT10 := L#85;
   MODE_LIST_RVS3[3060].DINT0 := L#16383;
   MODE_LIST_RVS3[3060].DINT1 := L#-16;
   MODE_LIST_RVS3[3060].DINT2 := L#-10944;
   MODE_LIST_RVS3[3060].DINT3 := L#16383;
   MODE_LIST_RVS3[3060].DINT4 := L#3840;
   MODE_LIST_RVS3[3060].DINT5 := L#-10651712;
   MODE_LIST_RVS3[3060].DINT6 := L#2147483647;
   MODE_LIST_RVS3[3060].DINT7 := L#1048533;
   MODE_LIST_RVS3[3060].DINT8 := L#268369920;
   MODE_LIST_RVS3[3060].DINT9 := L#268374015;
   MODE_LIST_RVS3[3060].DINT10 := L#85;
   MODE_LIST_RVS3[3061].DINT0 := L#16383;
   MODE_LIST_RVS3[3061].DINT1 := L#-16;
   MODE_LIST_RVS3[3061].DINT2 := L#-10944;
   MODE_LIST_RVS3[3061].DINT3 := L#62463;
   MODE_LIST_RVS3[3061].DINT4 := L#15360;
   MODE_LIST_RVS3[3061].DINT5 := L#-10651712;
   MODE_LIST_RVS3[3061].DINT6 := L#2147483647;
   MODE_LIST_RVS3[3061].DINT7 := L#1048533;
   MODE_LIST_RVS3[3061].DINT8 := L#268369920;
   MODE_LIST_RVS3[3061].DINT9 := L#268374015;
   MODE_LIST_RVS3[3061].DINT10 := L#85;
   MODE_LIST_RVS3[3062].DINT0 := L#16383;
   MODE_LIST_RVS3[3062].DINT1 := L#-16;
   MODE_LIST_RVS3[3062].DINT2 := L#-10944;
   MODE_LIST_RVS3[3062].DINT3 := L#984063;
   MODE_LIST_RVS3[3062].DINT4 := L#245760;
   MODE_LIST_RVS3[3062].DINT5 := L#-10651712;
   MODE_LIST_RVS3[3062].DINT6 := L#2147483647;
   MODE_LIST_RVS3[3062].DINT7 := L#1048533;
   MODE_LIST_RVS3[3062].DINT8 := L#268369920;
   MODE_LIST_RVS3[3062].DINT9 := L#268374015;
   MODE_LIST_RVS3[3062].DINT10 := L#85;
   MODE_LIST_RVS3[3063].DINT0 := L#16383;
   MODE_LIST_RVS3[3063].DINT1 := L#-16;
   MODE_LIST_RVS3[3063].DINT2 := L#-10944;
   MODE_LIST_RVS3[3063].DINT3 := L#15729663;
   MODE_LIST_RVS3[3063].DINT4 := L#3932160;
   MODE_LIST_RVS3[3063].DINT5 := L#-10651712;
   MODE_LIST_RVS3[3063].DINT6 := L#2147483647;
   MODE_LIST_RVS3[3063].DINT7 := L#1048533;
   MODE_LIST_RVS3[3063].DINT8 := L#268369920;
   MODE_LIST_RVS3[3063].DINT9 := L#268374015;
   MODE_LIST_RVS3[3063].DINT10 := L#85;
   MODE_LIST_RVS3[3064].DINT0 := L#16383;
   MODE_LIST_RVS3[3064].DINT1 := L#-16;
   MODE_LIST_RVS3[3064].DINT2 := L#-10944;
   MODE_LIST_RVS3[3064].DINT3 := L#12583935;
   MODE_LIST_RVS3[3064].DINT4 := L#3145728;
   MODE_LIST_RVS3[3064].DINT5 := L#-10651712;
   MODE_LIST_RVS3[3064].DINT6 := L#2147483647;
   MODE_LIST_RVS3[3064].DINT7 := L#1048533;
   MODE_LIST_RVS3[3064].DINT8 := L#268369920;
   MODE_LIST_RVS3[3064].DINT9 := L#268374015;
   MODE_LIST_RVS3[3064].DINT10 := L#85;
   MODE_LIST_RVS3[3065].DINT0 := L#16383;
   MODE_LIST_RVS3[3065].DINT1 := L#-16;
   MODE_LIST_RVS3[3065].DINT2 := L#-10944;
   MODE_LIST_RVS3[3065].DINT3 := L#-1073740801;
   MODE_LIST_RVS3[3065].DINT4 := L#-268435441;
   MODE_LIST_RVS3[3065].DINT5 := L#-8521789;
   MODE_LIST_RVS3[3065].DINT6 := L#2147221504;
   MODE_LIST_RVS3[3065].DINT7 := L#1048533;
   MODE_LIST_RVS3[3065].DINT8 := L#268369920;
   MODE_LIST_RVS3[3065].DINT9 := L#268374015;
   MODE_LIST_RVS3[3065].DINT10 := L#85;
   MODE_LIST_RVS3[3066].DINT0 := L#16383;
   MODE_LIST_RVS3[3066].DINT1 := L#-16;
   MODE_LIST_RVS3[3066].DINT2 := L#-10944;
   MODE_LIST_RVS3[3066].DINT3 := L#1023;
   MODE_LIST_RVS3[3066].DINT4 := L#-1073741821;
   MODE_LIST_RVS3[3066].DINT5 := L#-8521792;
   MODE_LIST_RVS3[3066].DINT6 := L#2147221504;
   MODE_LIST_RVS3[3066].DINT7 := L#1048533;
   MODE_LIST_RVS3[3066].DINT8 := L#268369920;
   MODE_LIST_RVS3[3066].DINT9 := L#268374015;
   MODE_LIST_RVS3[3066].DINT10 := L#85;
   MODE_LIST_RVS3[3067].DINT0 := L#16383;
   MODE_LIST_RVS3[3067].DINT1 := L#-16;
   MODE_LIST_RVS3[3067].DINT2 := L#-10944;
   MODE_LIST_RVS3[3067].DINT3 := L#1023;
   MODE_LIST_RVS3[3067].DINT4 := L#240;
   MODE_LIST_RVS3[3067].DINT5 := L#-8521732;
   MODE_LIST_RVS3[3067].DINT6 := L#2147221504;
   MODE_LIST_RVS3[3067].DINT7 := L#1048533;
   MODE_LIST_RVS3[3067].DINT8 := L#268369920;
   MODE_LIST_RVS3[3067].DINT9 := L#268374015;
   MODE_LIST_RVS3[3067].DINT10 := L#85;
   MODE_LIST_RVS3[3068].DINT0 := L#16383;
   MODE_LIST_RVS3[3068].DINT1 := L#-16;
   MODE_LIST_RVS3[3068].DINT2 := L#-10944;
   MODE_LIST_RVS3[3068].DINT3 := L#1023;
   MODE_LIST_RVS3[3068].DINT5 := L#-8521792;
   MODE_LIST_RVS3[3068].DINT6 := L#2147221504;
   MODE_LIST_RVS3[3068].DINT7 := L#1048533;
   MODE_LIST_RVS3[3068].DINT8 := L#268369920;
   MODE_LIST_RVS3[3068].DINT9 := L#268374015;
   MODE_LIST_RVS3[3068].DINT10 := L#85;
   MODE_LIST_RVS3[3069].DINT0 := L#16383;
   MODE_LIST_RVS3[3069].DINT1 := L#-16;
   MODE_LIST_RVS3[3069].DINT2 := L#-10944;
   MODE_LIST_RVS3[3069].DINT3 := L#1023;
   MODE_LIST_RVS3[3069].DINT5 := L#-10651712;
   MODE_LIST_RVS3[3069].DINT6 := L#1568145407;
   MODE_LIST_RVS3[3069].DINT7 := L#1048533;
   MODE_LIST_RVS3[3069].DINT8 := L#268369920;
   MODE_LIST_RVS3[3069].DINT9 := L#268374015;
   MODE_LIST_RVS3[3069].DINT10 := L#85;
   MODE_LIST_RVS3[3070].DINT0 := L#16383;
   MODE_LIST_RVS3[3070].DINT1 := L#-16;
   MODE_LIST_RVS3[3070].DINT2 := L#-10944;
   MODE_LIST_RVS3[3070].DINT3 := L#1023;
   MODE_LIST_RVS3[3070].DINT5 := L#-10651712;
   MODE_LIST_RVS3[3070].DINT6 := L#2147483647;
   MODE_LIST_RVS3[3070].DINT7 := L#1048533;
   MODE_LIST_RVS3[3070].DINT8 := L#268369920;
   MODE_LIST_RVS3[3070].DINT9 := L#268374015;
   MODE_LIST_RVS3[3070].DINT10 := L#85;
   MODE_LIST_RVS3[3071].DINT0 := L#16383;
   MODE_LIST_RVS3[3071].DINT1 := L#-16;
   MODE_LIST_RVS3[3071].DINT2 := L#-10944;
   MODE_LIST_RVS3[3071].DINT3 := L#1023;
   MODE_LIST_RVS3[3071].DINT5 := L#-8521792;
   MODE_LIST_RVS3[3071].DINT6 := L#2147221504;
   MODE_LIST_RVS3[3071].DINT7 := L#16777173;
   MODE_LIST_RVS3[3071].DINT8 := L#268369980;
   MODE_LIST_RVS3[3071].DINT9 := L#268433245;
   MODE_LIST_RVS3[3071].DINT10 := L#85;
   MODE_LIST_RVS3[3072].DINT0 := L#16383;
   MODE_LIST_RVS3[3072].DINT1 := L#-16;
   MODE_LIST_RVS3[3072].DINT2 := L#-10944;
   MODE_LIST_RVS3[3072].DINT3 := L#1023;
   MODE_LIST_RVS3[3072].DINT5 := L#-8521792;
   MODE_LIST_RVS3[3072].DINT6 := L#2147221504;
   MODE_LIST_RVS3[3072].DINT7 := L#1048533;
   MODE_LIST_RVS3[3072].DINT8 := L#268370880;
   MODE_LIST_RVS3[3072].DINT9 := L#-144896001;
   MODE_LIST_RVS3[3072].DINT10 := L#85;
   MODE_LIST_RVS3[3073].DINT0 := L#16383;
   MODE_LIST_RVS3[3073].DINT1 := L#-16;
   MODE_LIST_RVS3[3073].DINT2 := L#-10944;
   MODE_LIST_RVS3[3073].DINT3 := L#1023;
   MODE_LIST_RVS3[3073].DINT5 := L#-8521792;
   MODE_LIST_RVS3[3073].DINT6 := L#2147221504;
   MODE_LIST_RVS3[3073].DINT7 := L#1007681493;
   MODE_LIST_RVS3[3073].DINT8 := L#268373760;
   MODE_LIST_RVS3[3073].DINT9 := L#-144896001;
   MODE_LIST_RVS3[3073].DINT10 := L#85;
   MODE_LIST_RVS3[3074].DINT0 := L#16383;
   MODE_LIST_RVS3[3074].DINT1 := L#-16;
   MODE_LIST_RVS3[3074].DINT2 := L#-10944;
   MODE_LIST_RVS3[3074].DINT3 := L#1023;
   MODE_LIST_RVS3[3074].DINT5 := L#-8521792;
   MODE_LIST_RVS3[3074].DINT6 := L#2147221504;
   MODE_LIST_RVS3[3074].DINT7 := L#-267386923;
   MODE_LIST_RVS3[3074].DINT8 := L#268385280;
   MODE_LIST_RVS3[3074].DINT9 := L#-144896001;
   MODE_LIST_RVS3[3074].DINT10 := L#85;
   MODE_LIST_RVS3[3075].DINT0 := L#16383;
   MODE_LIST_RVS3[3075].DINT1 := L#-16;
   MODE_LIST_RVS3[3075].DINT2 := L#-10944;
   MODE_LIST_RVS3[3075].DINT3 := L#1023;
   MODE_LIST_RVS3[3075].DINT5 := L#-8521792;
   MODE_LIST_RVS3[3075].DINT6 := L#2147221504;
   MODE_LIST_RVS3[3075].DINT7 := L#-1072693291;
   MODE_LIST_RVS3[3075].DINT8 := L#268431363;
   MODE_LIST_RVS3[3075].DINT9 := L#-144896001;
   MODE_LIST_RVS3[3075].DINT10 := L#85;
   MODE_LIST_RVS3[3076].DINT0 := L#16383;
   MODE_LIST_RVS3[3076].DINT1 := L#-16;
   MODE_LIST_RVS3[3076].DINT2 := L#-10944;
   MODE_LIST_RVS3[3076].DINT3 := L#1023;
   MODE_LIST_RVS3[3076].DINT5 := L#-8521792;
   MODE_LIST_RVS3[3076].DINT6 := L#2147221504;
   MODE_LIST_RVS3[3076].DINT7 := L#-1072693291;
   MODE_LIST_RVS3[3076].DINT8 := L#268431363;
   MODE_LIST_RVS3[3076].DINT9 := L#-144896001;
   MODE_LIST_RVS3[3076].DINT10 := L#85;
   MODE_LIST_RVS3[3077].DINT0 := L#16383;
   MODE_LIST_RVS3[3077].DINT1 := L#-16;
   MODE_LIST_RVS3[3077].DINT2 := L#-10944;
   MODE_LIST_RVS3[3077].DINT3 := L#1023;
   MODE_LIST_RVS3[3077].DINT5 := L#-8521792;
   MODE_LIST_RVS3[3077].DINT6 := L#2147221504;
   MODE_LIST_RVS3[3077].DINT7 := L#1048533;
   MODE_LIST_RVS3[3077].DINT8 := L#-144900096;
   MODE_LIST_RVS3[3077].DINT9 := L#268371805;
   MODE_LIST_RVS3[3077].DINT10 := L#85;
   MODE_LIST_RVS3[3078].DINT0 := L#16383;
   MODE_LIST_RVS3[3078].DINT1 := L#-16;
   MODE_LIST_RVS3[3078].DINT2 := L#-10944;
   MODE_LIST_RVS3[3078].DINT3 := L#1023;
   MODE_LIST_RVS3[3078].DINT5 := L#-8521792;
   MODE_LIST_RVS3[3078].DINT6 := L#2147221504;
   MODE_LIST_RVS3[3078].DINT7 := L#1048533;
   MODE_LIST_RVS3[3078].DINT8 := L#268369920;
   MODE_LIST_RVS3[3078].DINT9 := L#268433245;
   MODE_LIST_RVS3[3078].DINT10 := L#85;
   MODE_LIST_RVS3[3079].DINT0 := L#16383;
   MODE_LIST_RVS3[3079].DINT1 := L#-16;
   MODE_LIST_RVS3[3079].DINT2 := L#-10944;
   MODE_LIST_RVS3[3079].DINT3 := L#1023;
   MODE_LIST_RVS3[3079].DINT5 := L#-8521792;
   MODE_LIST_RVS3[3079].DINT6 := L#2147221504;
   MODE_LIST_RVS3[3079].DINT7 := L#1048533;
   MODE_LIST_RVS3[3079].DINT8 := L#268369920;
   MODE_LIST_RVS3[3079].DINT9 := L#-144896001;
   MODE_LIST_RVS3[3079].DINT10 := L#85;
END_DATA_BLOCK

DATA_BLOCK DB 5002
VERSION : 0.0
"从端与主端通讯"
BEGIN
END_DATA_BLOCK

DATA_BLOCK "MAIN_ToHMI"	// DB 6002
VERSION : 0.1
  STRUCT
   SDPF_B_ToHMI : WORD ;
   SDPF_B_PFB : REAL ;
   SDPF_K1_B1_ToHMI : WORD ;
   SDPF_K1_B1_PFB : REAL ;
   SDPF_K2_B1_ToHMI : WORD ;
   SDPF_K2_B1_PFB : REAL ;
   SDPF_K3_B1_ToHMI : WORD ;
   SDPF_K3_B1_PFB : REAL ;
   SDPF_YL_ToHMI : WORD ;
   SDPF_YL_PFB : REAL ;
   AP_PSB_A_ToHMI : WORD ;
   AP_PSB_A_Level : INT ;
   AP_PSB_D_ToHMI : WORD ;
   AP_PSB_D_Level : INT ;
   AP_JPB_1_ToHMI : WORD ;
   AP_JPB_1_Level : INT ;
   AP_FSB_1_ToHMI : WORD ;
   AP_FSB_1_Level : INT ;
   AP_WSB_ToHMI : WORD ;
   AP_WSB_Level : INT ;
   LQSB_ToHMI : WORD ;
   LQSB_Level : INT ;
   AT_BYSB1_ToHMI1 : WORD ;
   AT_BYSB1_ToHMI2 : WORD ;
   AT_BYSB1_Level : INT ;
   AT_BYSB1_RT : REAL ;
   AT_BYSB1_FltNo : INT ;
   AT_BYSB2_ToHMI1 : WORD ;
   AT_BYSB2_ToHMI2 : WORD ;
   AT_BYSB2_Level : INT ;
   AT_BYSB2_RT : REAL ;
   AT_BYSB2_FltNo : INT ;
   AT_BYSB3_ToHMI1 : WORD ;
   AT_BYSB3_ToHMI2 : WORD ;
   AT_BYSB3_Level : INT ;
   AT_BYSB3_RT : REAL ;
   AT_BYSB3_FltNo : INT ;
   AT_BYSB4_ToHMI1 : WORD ;
   AT_BYSB4_ToHMI2 : WORD ;
   AT_BYSB4_Level : INT ;
   AT_BYSB4_RT : REAL ;
   AT_BYSB4_FltNo : INT ;
   AT_FSB_ToHMI1 : WORD ;
   AT_FSB_ToHMI2 : WORD ;
   AT_FSB_Level : INT ;
   AT_FSB_RT : REAL ;
   AT_FSB_FltNo : INT ;
   AP_PSB_ToHMI1 : WORD ;
   AP_PSB_ToHMI2 : WORD ;
   AP_PSB_Level : INT ;
   AP_PSB_RT : REAL ;
   AP_PSB_FltNo : INT ;
   YL_YSB_ToHMI1 : WORD ;
   YL_YSB_ToHMI2 : WORD ;
   YL_YSB_Level : INT ;
   YL_YSB_RT : REAL ;
   YL_YSB_FltNo : INT ;
   C_B1_CO2 : REAL ;
   C_B2_CO2 : REAL ;
   C_B3_CO2 : REAL ;
   C_B4_CO2 : REAL ;
   C_A1_CO2 : REAL ;
   YL_CO2 : REAL ;
   H_B5_Humi : REAL ;
   H_B5_Temp : REAL ;
   H_B4_Humi : REAL ;
   H_B4_Temp : REAL ;
   K3_T_B1_Humi : REAL ;
   K3_T_B1_Temp : REAL ;
   K1_T_B3_Humi : REAL ;
   K1_T_B3_Temp : REAL ;
   K1_T_B2_Humi : REAL ;
   K1_T_B2_Temp : REAL ;
   K1_T_B5_Humi : REAL ;
   K1_T_B5_Temp : REAL ;
   T_B1_Humi : REAL ;
   T_B1_Temp : REAL ;
   T_B2_Humi : REAL ;
   T_B2_Temp : REAL ;
   K1_T_B1_Humi : REAL ;
   K1_T_B1_Temp : REAL ;
   K1_T_B4_Humi : REAL ;
   K1_T_B4_Temp : REAL ;
   K2_H_B1_Humi : REAL ;
   K2_H_B1_Temp : REAL ;
   H_B2_Humi : REAL ;
   H_B2_Temp : REAL ;
   H_B3_Humi : REAL ;
   H_B3_Temp : REAL ;
   K2_T_B1_Humi : REAL ;
   K2_T_B1_Temp : REAL ;
   H_B6_Humi : REAL ;
   H_B6_Temp : REAL ;
   H_B7_Humi : REAL ;
   H_B7_Temp : REAL ;
   K3_H_B1_Humi : REAL ;
   K3_H_B1_Temp : REAL ;
   K1_H_B1_Humi : REAL ;
   K1_H_B1_Temp : REAL ;
   H_B1_Humi : REAL ;
   H_B1_Temp : REAL ;
   T_A1_Humi : REAL ;
   T_A1_Temp : REAL ;
   K1_T_B6_Humi : REAL ;
   K1_T_B6_Temp : REAL ;
   YL_TH6_Humi : REAL ;
   YL_TH6_Temp : REAL ;
   KT_B1_ToHMI1 : WORD ;
   KT_B1_ToHMI2 : WORD ;
   KT_B1_VFRT : DWORD ;
   KT_B1_RPM : INT ;
   KT_B1_MotrCurr : INT ;
   KT_B1_AxleT : INT ;
   KT_B1_WindT : INT ;
   KT_B1_VFFB : INT ;
   KT_B1_RealTP : INT ;
   KT_B1_ECSum : DWORD ;
   KT_B1_FltNo : INT ;
   KT_B1_RT : REAL ;
   YL_KT_B1_1 : WORD ;
   YL_KT_B1_2 : WORD ;
   YL_KT_B1_3 : WORD ;
   YL_KT_B1_4 : WORD ;
   HPF_B1_ToHMI1 : WORD ;
   HPF_B1_ToHMI2 : WORD ;
   HPF_B1_VFFB : INT ;
   HPF_B1_A_Pcurr : INT ;
   HPF_B1_B_Pcurr : INT ;
   HPF_B1_C_Pcurr : INT ;
   HPF_B1_A_Pvolt : INT ;
   HPF_B1_B_Pvolt : INT ;
   HPF_B1_C_Pvolt : INT ;
   HPF_B1_RT : REAL ;
   HPF_B1_FltNo : INT ;
   YL_HPF_B1_1 : WORD ;
   YL_HPF_B1_2 : WORD ;
   YL_HPF_B1_3 : WORD ;
   YL_HPF_B1_4 : WORD ;
   UOF_B1_ToHMI1 : WORD ;
   UOF_B1_ToHMI2 : WORD ;
   UOF_B1_VFFB : INT ;
   UOF_B1_A_Pcurr : INT ;
   UOF_B1_B_Pcurr : INT ;
   UOF_B1_C_Pcurr : INT ;
   UOF_B1_A_Pvolt : INT ;
   UOF_B1_B_Pvolt : INT ;
   UOF_B1_C_Pvolt : INT ;
   UOF_B1_FAxleT : INT ;
   UOF_B1_RAxleT : INT ;
   UOF_B1_A_WindT : INT ;
   UOF_B1_B_WindT : INT ;
   UOF_B1_C_WindT : INT ;
   UOF_B1_H_Vibr : INT ;
   UOF_B1_V_Vibr : INT ;
   UOF_B1_RT : REAL ;
   UOF_B1_FltNo : INT ;
   YL_UOF_B1_1 : WORD ;
   YL_UOF_B1_2 : WORD ;
   YL_UOF_B1_3 : WORD ;
   YL_UOF_B1_4 : WORD ;
   TVF_B1_ToHMI1 : WORD ;
   TVF_B1_ToHMI2 : WORD ;
   TVF_B1_A_Pcurr : INT ;
   TVF_B1_B_Pcurr : INT ;
   TVF_B1_C_Pcurr : INT ;
   TVF_B1_A_Pvolt : INT ;
   TVF_B1_B_Pvolt : INT ;
   TVF_B1_C_Pvolt : INT ;
   TVF_B1_FAxleT : INT ;
   TVF_B1_RAxleT : INT ;
   TVF_B1_A_WindT : INT ;
   TVF_B1_B_WindT : INT ;
   TVF_B1_C_WindT : INT ;
   TVF_B1_X_Vibr : INT ;
   TVF_B1_Y_Vibr : INT ;
   TVF_B1_RT : REAL ;
   TVF_B1_FltNo : INT ;
   YL_TVF_B1_1 : WORD ;
   YL_TVF_B1_2 : WORD ;
   YL_TVF_B1_3 : WORD ;
   YL_TVF_B1_4 : WORD ;
   TVF_B2_ToHMI1 : WORD ;
   TVF_B2_ToHMI2 : WORD ;
   TVF_B2_A_Pcurr : INT ;
   TVF_B2_B_Pcurr : INT ;
   TVF_B2_C_Pcurr : INT ;
   TVF_B2_A_Pvolt : INT ;
   TVF_B2_B_Pvolt : INT ;
   TVF_B2_C_Pvolt : INT ;
   TVF_B2_FAxleT : INT ;
   TVF_B2_RAxleT : INT ;
   TVF_B2_A_WindT : INT ;
   TVF_B2_B_WindT : INT ;
   TVF_B2_C_WindT : INT ;
   TVF_B2_H_Vibr : INT ;
   TVF_B2_V_Vibr : INT ;
   TVF_B2_RT : REAL ;
   TVF_B2_FltNo : INT ;
   YL_TVF_B2_1 : WORD ;
   YL_TVF_B2_2 : WORD ;
   YL_TVF_B2_3 : WORD ;
   YL_TVF_B2_4 : WORD ;
   SK1_DTS_B1_ToHMI : WORD ;
   SK1_DTS_B2_ToHMI : WORD ;
   SK1_DTS_B3_ToHMI : WORD ;
   SK2_DTS_B1_ToHMI : WORD ;
   SK2_DTS_B2_ToHMI : WORD ;
   SK2_DTS_B3_ToHMI : WORD ;
   SK3_DTS_B1_ToHMI : WORD ;
   SK3_DTS_B2_ToHMI : WORD ;
   SK3_DTS_B3_ToHMI : WORD ;
   ST1_D_B1_ToHMI : WORD ;
   ST1_D_B2_ToHMI : WORD ;
   ST4_D_B1_ToHMI : WORD ;
   ST5_D_B1_ToHMI : WORD ;
   YL_D_1 : WORD ;
   YL_D_2 : WORD ;
   YL_D_3 : WORD ;
   YL_D_4 : WORD ;
   YL_D_5 : WORD ;
   SDM_B1_ToHMI : WORD ;
   SDM_B2_ToHMI : WORD ;
   SDM_B3_ToHMI : WORD ;
   SDM_B4_ToHMI : WORD ;
   SDM_B5_ToHMI : WORD ;
   SDM_B6_ToHMI : WORD ;
   SDM_B7_ToHMI : WORD ;
   SDM_B8_ToHMI : WORD ;
   SUOF_DT_B1_ToHMI : WORD ;
   SUOF_DT_B2_ToHMI : WORD ;
   SUOF_DT_B3_ToHMI : WORD ;
   SUOF_DT_B4_ToHMI : WORD ;
   YL_DT_1 : WORD ;
   YL_DT_2 : WORD ;
   YL_DT_3 : WORD ;
   YL_DT_4 : WORD ;
   YL_DT_5 : WORD ;
   SDTS_B1_ToHMI : WORD ;
   SDTS_B2_ToHMI : WORD ;
   SDTS_B3_ToHMI : WORD ;
   SDTS_B4_ToHMI : WORD ;
   SDTS_B5_ToHMI : WORD ;
   SDTS_B6_ToHMI : WORD ;
   SDT_RFS_B1_ToHMI : WORD ;
   T1_XSF_B1_ToHMI : WORD ;
   T1_XSF_B1_A_Pcurr : INT ;
   T1_XSF_B1_B_Pcurr : INT ;
   T1_XSF_B1_C_Pcurr : INT ;
   T1_XSF_B1_RT : REAL ;
   T1_XSF_B1_FltNo : INT ;
   RFP_B_ToHMI : WORD ;
   RFP_B_A_Pcurr : INT ;
   RFP_B_B_Pcurr : INT ;
   RFP_B_C_Pcurr : INT ;
   RFP_B_RT : REAL ;
   RFP_B_FltNo : INT ;
   K1_HPF_B1_ToHMI : WORD ;
   K1_HPF_B1_A_Pcurr : INT ;
   K1_HPF_B1_B_Pcurr : INT ;
   K1_HPF_B1_C_Pcurr : INT ;
   K1_HPF_B1_RT : REAL ;
   K1_HPF_B1_FltNo : INT ;
   K2_HPF_B1_ToHMI : WORD ;
   K2_HPF_B1_A_Pcurr : INT ;
   K2_HPF_B1_B_Pcurr : INT ;
   K2_HPF_B1_C_Pcurr : INT ;
   K2_HPF_B1_RT : REAL ;
   K2_HPF_B1_FltNo : INT ;
   K3_HPF_B1_ToHMI : WORD ;
   K3_HPF_B1_A_Pcurr : INT ;
   K3_HPF_B1_B_Pcurr : INT ;
   K3_HPF_B1_C_Pcurr : INT ;
   K3_HPF_B1_RT : REAL ;
   K3_HPF_B1_FltNo : INT ;
   T5_XPF_B1_ToHMI : WORD ;
   T5_XPF_B1_A_Pcurr : INT ;
   T5_XPF_B1_B_Pcurr : INT ;
   T5_XPF_B1_C_Pcurr : INT ;
   T5_XPF_B1_RT : REAL ;
   T5_XPF_B1_FltNo : INT ;
   T1_XPF_B1_ToHMI : WORD ;
   T1_XPF_B1_A_Pcurr : INT ;
   T1_XPF_B1_B_Pcurr : INT ;
   T1_XPF_B1_C_Pcurr : INT ;
   T1_XPF_B1_RT : REAL ;
   T1_XPF_B1_FltNo : INT ;
   T4_XPF_B1_ToHMI : WORD ;
   T4_XPF_B1_A_Pcurr : INT ;
   T4_XPF_B1_B_Pcurr : INT ;
   T4_XPF_B1_C_Pcurr : INT ;
   T4_XPF_B1_RT : REAL ;
   T4_XPF_B1_FltNo : INT ;
   K1_XK_B1_ToHMI : WORD ;
   K1_XK_B1_A_Pcurr : INT ;
   K1_XK_B1_B_Pcurr : INT ;
   K1_XK_B1_C_Pcurr : INT ;
   K1_XK_B1_RT : REAL ;
   K1_XK_B1_FltNo : INT ;
   K2_XK_B2_ToHMI : WORD ;
   K2_XK_B2_A_Pcurr : INT ;
   K2_XK_B2_B_Pcurr : INT ;
   K2_XK_B2_C_Pcurr : INT ;
   K2_XK_B2_RT : REAL ;
   K2_XK_B2_FltNo : INT ;
   K3_XK_B3_ToHMI : WORD ;
   K3_XK_B3_A_Pcurr : INT ;
   K3_XK_B3_B_Pcurr : INT ;
   K3_XK_B3_C_Pcurr : INT ;
   K3_XK_B3_RT : REAL ;
   K3_XK_B3_FltNo : INT ;
   YL_IMCC_FJ_1_ToHMI : WORD ;
   YL_IMCC_FJ_1_Pcurr : INT ;
   YL_IMCC_FJ_1_RunTime : REAL ;
   YL_IMCC_FJ_1_FltNo : INT ;
   YL_IMCC_FJ_2_ToHMI : WORD ;
   YL_IMCC_FJ_2_Pcurr : INT ;
   YL_IMCC_FJ_2_RunTime : REAL ;
   YL_IMCC_FJ_2_FltNo : INT ;
   YL_IMCC_FJ_3_ToHMI : WORD ;
   YL_IMCC_FJ_3_Pcurr : INT ;
   YL_IMCC_FJ_3_RunTime : REAL ;
   YL_IMCC_FJ_3_FltNo : INT ;
   YL_IMCC_FJ_4_ToHMI : WORD ;
   YL_IMCC_FJ_4_Pcurr : INT ;
   YL_IMCC_FJ_4_RunTime : REAL ;
   YL_IMCC_FJ_4_FltNo : INT ;
   YL_IMCC_FJ_5_ToHMI : WORD ;
   YL_IMCC_FJ_5_Pcurr : INT ;
   YL_IMCC_FJ_5_RunTime : REAL ;
   YL_IMCC_FJ_5_FltNo : INT ;
   RFM_ToHMI : WORD ;
   JH_YC_B_ToHMI : WORD ;
   E420_02_N_ToHMI : WORD ;
   E420_03_N_ToHMI : WORD ;
   E420_04_K_ToHMI : WORD ;
   E420_08_K_ToHMI : WORD ;
   YL_FT1_ToHMI : WORD ;
   YL_FT2_ToHMI : WORD ;
   YL_FT3_ToHMI : WORD ;
   YL_FT4_ToHMI : WORD ;
   H420_02_K_ToHMI : WORD ;
   H420_02_K_FLOOR : WORD ;
   systemStatus : ARRAY  [0 .. 5 ] OF WORD ;
   firstUnitStatus : ARRAY  [0 .. 15 ] OF WORD ;
   secondUnitStatus : ARRAY  [0 .. 15 ] OF WORD ;
   thirdUnitStatus : ARRAY  [0 .. 15 ] OF WORD ;
   EPS22_ToHMI1 : WORD ;
   EPS22_ToHMI : ARRAY  [0 .. 15 ] OF INT  := 0;
   EPS12_ToHMI1 : WORD ;
   EPS12_ToHMI : ARRAY  [0 .. 15 ] OF INT ;
   ZNZM_abd3 : WORD ;
   VRV_ToHMI : ARRAY  [0 .. 20 ] OF WORD  := W#16#0;
   VRV_ToHMI1 : WORD ;
   WLE_1_ToHMI : WORD ;
   WLE_2_ToHMI : WORD ;
   WLE_3_ToHMI : WORD ;
   WLE_4_ToHMI : WORD ;
   XFDF_B1_TOHMI : WORD ;
   XFDF_B2_TOHMI : WORD ;
   IMCC_Com_B : WORD ;
  END_STRUCT ;	
BEGIN
END_DATA_BLOCK

DATA_BLOCK "ISCS_CONTROL"	// DB 6003
VERSION : 0.1
  STRUCT
   DPH_K4_A1_SCtrl : WORD ;
   DPH_A_SCtrl : WORD ;
   DPF_YL_SCtrl : WORD ;
   DPF_YL1_SCtrl : WORD ;
   AT_AYSB1_SCtrl : WORD ;
   AT_AYSB2_SCtrl : WORD ;
   AT_AYSB3_SCtrl : WORD ;
   AT_AYSB4_SCtrl : WORD ;
   AT_QJFSB_SCtrl : WORD ;
   AT_FSB_SCtrl : WORD ;
   AT_YL_SCtrl : WORD ;
   KT_A1_SCtrl : WORD ;
   HPF_A1_SCtrl : WORD ;
   UOF_A1_SCtrl : WORD ;
   TVF_A1_SCtrl : WORD ;
   TVF_A2_SCtrl : WORD ;
   K4_DTS_A1_SCtrl : WORD ;
   K4_DTS_A2_SCtrl : WORD ;
   K4_DTS_A3_SCtrl : WORD ;
   DTS_A1_SCtrl : WORD ;
   DTS_A2_SCtrl : WORD ;
   DTS_A3_SCtrl : WORD ;
   DTS_A4_SCtrl : WORD ;
   DTS_A5_SCtrl : WORD ;
   DTS_A6_SCtrl : WORD ;
   DT_RFS_A1_SCtrl : WORD ;
   T6_D_A1_SCtrl : WORD ;
   T6_D_A2_SCtrl : WORD ;
   T7_D_A1_SCtrl : WORD ;
   DM_A1_SCtrl : WORD ;
   DM_A2_SCtrl : WORD ;
   DM_A3_SCtrl : WORD ;
   DM_A4_SCtrl : WORD ;
   DM_A5_SCtrl : WORD ;
   DM_A6_SCtrl : WORD ;
   DM_A7_SCtrl : WORD ;
   DM_A8_SCtrl : WORD ;
   U0F_DT_A1_SCtrl : WORD ;
   U0F_DT_A2_SCtrl : WORD ;
   U0F_DT_A3_SCtrl : WORD ;
   U0F_DT_A4_SCtrl : WORD ;
   YL_D_1 : WORD ;
   YL_D_2 : WORD ;
   YL_DT_1 : WORD ;
   YL_DT_2 : WORD ;
   RFS_A1_SCtrl : WORD ;
   T6_XSF_A1_SCtrl : WORD ;
   T6_XPF_A1_SCtrl : WORD ;
   T7_XPF_A1_SCtrl : WORD ;
   K4_XK_A1_SCtrl : WORD ;
   K4_HPF_A1_SCtrl : WORD ;
   WLE_1_SCtrl : WORD ;
   WLE_2_SCtrl : WORD ;
   WLE_3_SCtrl : WORD ;
   WLE_4_SCtrl : WORD ;
   YL_DATA : ARRAY  [0 .. 151 ] OF WORD ;
   KT_A1_KpTm : INT ;
   KT_A1_KiTm : INT ;
   KT_A1_SPTm : INT ;
   KT_A1_OMS : INT ;
   HPF_A1_KpTm : INT ;
   HPF_A1_KiTm : INT ;
   HPF_A1_SPTm : INT ;
   HPF_A1_OMS : INT ;
   UOF_A1_KpTm : INT ;
   UOF_A1_KiTm : INT ;
   UOF_A1_SPTm : INT ;
   UOF_A1_OMS : INT ;
   DPF_K4_A1_KpTm : INT ;
   DPF_K4_A1_KiTm : INT ;
   DPF_K4_A1_SPTm : INT ;
   DPF_K4_A1_OMS : INT ;
   DPF_A_KpTm : INT ;
   DPF_A_KiTm : INT ;
   DPF_A_SPTm : INT ;
   DPF_A_OMS : INT ;
  END_STRUCT ;	
BEGIN
END_DATA_BLOCK

DATA_BLOCK "SLAVE_TO_HMI"	// DB 6004
VERSION : 0.1
  STRUCT
   DPF_A_ToHMI : WORD ;
   DPF_A_PFB : REAL ;
   DPF_K4_A1_ToHMI : WORD ;
   DPF_K4_A1_PFB : REAL ;
   DPF_YL_ToHMI : WORD ;
   DPF_YL_PFB : REAL ;
   AP_BMPSB_ToHMI : WORD ;
   AP_BMPSB_Level : INT ;
   AP_PSB_B_ToHMI : WORD ;
   AP_PSB_B_Level : INT ;
   AP_PSB_C_ToHMI : WORD ;
   AP_PSB_C_Level : INT ;
   AP_FSB_2_ToHMI : WORD ;
   AP_FSB_2_Level : INT ;
   YL_FSB_ToHMI : WORD ;
   YL_FSB_Level : INT ;
   AT_AYSB1_ToHMI1 : WORD ;
   AT_AYSB1_ToHMI2 : WORD ;
   AT_AYSB1_Level : INT ;
   AT_AYSB1_RT : REAL ;
   AT_AYSB1_FltNo : INT ;
   AT_AYSB2_ToHMI1 : WORD ;
   AT_AYSB2_ToHMI2 : WORD ;
   AT_AYSB2_Level : INT ;
   AT_AYSB2_RT : REAL ;
   AT_AYSB2_FltNo : INT ;
   AT_AYSB3_ToHMI1 : WORD ;
   AT_AYSB3_ToHMI2 : WORD ;
   AT_AYSB3_Level : INT ;
   AT_AYSB3_RT : REAL ;
   AT_AYSB3_FltNo : INT ;
   AT_AYSB4_ToHMI1 : WORD ;
   AT_AYSB4_ToHMI2 : WORD ;
   AT_AYSB4_Level : INT ;
   AT_AYSB4_RT : REAL ;
   AT_AYSB4_FltNo : INT ;
   YL_FSB1_ToHMI1 : WORD ;
   YL_FSB1_ToHMI2 : WORD ;
   YL_FSB1_Level : INT ;
   YL_FSB1_RT : REAL ;
   YL_FSB1_FltNo : INT ;
   AT_QJFSB_ToHMI1 : WORD ;
   AT_QJFSB_ToHMI2 : WORD ;
   AT_QJFSB_Level : INT ;
   AT_QJFSB_RT : REAL ;
   AT_QJFSB_FltNo : INT ;
   AT_FSB_ToHMI1 : WORD ;
   AT_FSBToHMI2 : WORD ;
   AT_FSB_Level : INT ;
   AT_FSB_RT : REAL ;
   AT_FSB_FltNo : INT ;
   YL_YSB1_ToHMI1 : WORD ;
   YL_YSB1_ToHMI2 : WORD ;
   YL_YSB1_Level : INT ;
   YL_YSB1_RT : REAL ;
   YL_YSB1_FltNo : INT ;
   C_A2_CO2 : REAL ;
   C_A3_CO2 : REAL ;
   C_A4_CO2 : REAL ;
   YL_CO2 : REAL ;
   H_A1_Humi : REAL ;
   H_A1_Temp : REAL ;
   K4_H_A1_Humi : REAL ;
   K4_H_A1_Temp : REAL ;
   H_A3_Humi : REAL ;
   H_A3_Temp : REAL ;
   H_A2_Humi : REAL ;
   H_A2_Temp : REAL ;
   K4_T_A1_Humi : REAL ;
   K4_T_A1_Temp : REAL ;
   H_A4_Humi : REAL ;
   H_A4_Temp : REAL ;
   H_A5_Humi : REAL ;
   H_A5_Temp : REAL ;
   H_A7_Humi : REAL ;
   H_A7_Temp : REAL ;
   H_A6_Humi : REAL ;
   H_A6_Temp : REAL ;
   T_A2_Humi : REAL ;
   T_A2_Temp : REAL ;
   YL_TH1_Humi : REAL ;
   YL_TH1_Temp : REAL ;
   YL_TH2_Humi : REAL ;
   YL_TH2_Temp : REAL ;
   YL_TH3_Humi : REAL ;
   YL_TH3_Temp : REAL ;
   YL_TH4_Humi : REAL ;
   YL_TH4_Temp : REAL ;
   YL_TH5_Humi : REAL ;
   YL_TH5_Temp : REAL ;
   YL_TH6_Humi : REAL ;
   YL_TH6_Temp : REAL ;
   KT_A1_ToHMI1 : WORD ;
   KT_A1_ToHMI2 : WORD ;
   KT_A1_VFRT : DWORD ;
   KT_A1_RPM : INT ;
   KT_A1_MotrCurr : INT ;
   KT_A1_AxleT : INT ;
   KT_A1_WindT : INT ;
   KT_A1_VFFB : INT ;
   KT_A1_RealTP : INT ;
   KT_A1_ECSum : DWORD ;
   KT_A1_FltNo : INT ;
   KT_A1_RT : REAL ;
   YL_KT_A1_1 : WORD ;
   YL_KT_A1_2 : WORD ;
   YL_KT_A1_3 : WORD ;
   YL_KT_A1_4 : WORD ;
   HPF_A1_ToHMI1 : WORD ;
   HPF_A1_ToHMI2 : WORD ;
   HPF_A1_VFFB : INT ;
   HPF_A1_A_Pcurr : INT ;
   HPF_A1_B_Pcurr : INT ;
   HPF_A1_C_Pcurr : INT ;
   HPF_A1_A_Pvolt : INT ;
   HPF_A1_B_Pvolt : INT ;
   HPF_A1_C_Pvolt : INT ;
   HPF_A1_RT : REAL ;
   HPF_A1_FltNo : INT ;
   YL_HPF_A1_1 : WORD ;
   YL_HPF_A1_2 : WORD ;
   YL_HPF_A1_3 : WORD ;
   YL_HPF_A1_4 : WORD ;
   UOF_A1_ToHMI1 : WORD ;
   UOF_A1_ToHMI2 : WORD ;
   UOF_A1_VFFB : INT ;
   UOF_A1_A_Pcurr : INT ;
   UOF_A1_B_Pcurr : INT ;
   UOF_A1_C_Pcurr : INT ;
   UOF_A1_A_Pvolt : INT ;
   UOF_A1_B_Pvolt : INT ;
   UOF_A1_C_Pvolt : INT ;
   UOF_A1_FAxleT : INT ;
   UOF_A1_RAxleT : INT ;
   UOF_A1_A_WindT : INT ;
   UOF_A1_B_WindT : INT ;
   UOF_A1_C_WindT : INT ;
   UOF_A1_H_Vibr : INT ;
   UOF_A1_V_Vibr : INT ;
   UOF_A1_RT : REAL ;
   UOF_A1_FltNo : INT ;
   YL_UOF_A1_1 : WORD ;
   YL_UOF_A1_2 : WORD ;
   YL_UOF_A1_3 : WORD ;
   YL_UOF_A1_4 : WORD ;
   TVF_A1_ToHMI1 : WORD ;
   TVF_A1_ToHMI2 : WORD ;
   TVF_A1_A_Pcurr : INT ;
   TVF_A1_B_Pcurr : INT ;
   TVF_A1_C_Pcurr : INT ;
   TVF_A1_A_Pvolt : INT ;
   TVF_A1_B_Pvolt : INT ;
   TVF_A1_C_Pvolt : INT ;
   TVF_A1_FAxleT : INT ;
   TVF_A1_RAxleT : INT ;
   TVF_A1_A_WindT : INT ;
   TVF_A1_B_WindT : INT ;
   TVF_A1_C_WindT : INT ;
   TVF_A1_X_Vibr : INT ;
   TVF_A1_Y_Vibr : INT ;
   TVF_A1_RT : REAL ;
   TVF_A1_FltNo : INT ;
   YL_TVF_A1_1 : WORD ;
   YL_TVF_A1_2 : WORD ;
   YL_TVF_A1_3 : WORD ;
   YL_TVF_A1_4 : WORD ;
   TVF_A2_ToHMI1 : WORD ;
   TVF_A2_ToHMI2 : WORD ;
   TVF_A2_A_Pcurr : INT ;
   TVF_A2_B_Pcurr : INT ;
   TVF_A2_C_Pcurr : INT ;
   TVF_A2_A_Pvolt : INT ;
   TVF_A2_B_Pvolt : INT ;
   TVF_A2_C_Pvolt : INT ;
   TVF_A2_FAxleT : INT ;
   TVF_A2_RAxleT : INT ;
   TVF_A2_A_WindT : INT ;
   TVF_A2_B_WindT : INT ;
   TVF_A2_C_WindT : INT ;
   TVF_A2_H_Vibr : INT ;
   TVF_A2_V_Vibr : INT ;
   TVF_A2_RT : REAL ;
   TVF_A2_FltNo : INT ;
   YL_TVF_A2_1 : WORD ;
   YL_TVF_A2_2 : WORD ;
   YL_TVF_A2_3 : WORD ;
   YL_TVF_A2_4 : WORD ;
   K4_DTS_A1_ToHMI : WORD ;
   K4_DTS_A2_ToHMI : WORD ;
   K4_DTS_A3_ToHMI : WORD ;
   T6_D_A1_ToHMI : WORD ;
   T6_D_A2_ToHMI : WORD ;
   T7_D_A1_ToHMI : WORD ;
   DM_A1_ToHMI : WORD ;
   DM_A2_ToHMI : WORD ;
   DM_A3_ToHMI : WORD ;
   DM_A4_ToHMI : WORD ;
   DM_A5_ToHMI : WORD ;
   DM_A6_ToHMI : WORD ;
   DM_A7_ToHMI : WORD ;
   DM_A8_ToHMI : WORD ;
   UOF_DT_A1_ToHMI : WORD ;
   UOF_DT_A2_ToHMI : WORD ;
   UOF_DT_A3_ToHMI : WORD ;
   UOF_DT_A4_ToHMI : WORD ;
   DTS_A1_ToHMI : WORD ;
   DTS_A2_ToHMI : WORD ;
   DTS_A3_ToHMI : WORD ;
   DTS_A4_ToHMI : WORD ;
   DTS_A5_ToHMI : WORD ;
   DTS_A6_ToHMI : WORD ;
   DT_RFS_A1_ToHMI : WORD ;
   YL_D_1 : WORD ;
   YL_D_2 : WORD ;
   YL_D_3 : WORD ;
   YL_D_4 : WORD ;
   YL_D_5 : WORD ;
   YL_DT_1 : WORD ;
   YL_DT_2 : WORD ;
   YL_DT_3 : WORD ;
   YL_DT_4 : WORD ;
   YL_DT_5 : WORD ;
   T6_XSF_A1_ToHMI : WORD ;
   T6_XSF_A1_A_Pcurr : INT ;
   T6_XSF_A1_B_Pcurr : INT ;
   T6_XSF_A1_C_Pcurr : INT ;
   T6_XSF_A1_RT : REAL ;
   T6_XSF_A1_FltNo : INT ;
   RFS_A_ToHMI : WORD ;
   RFS_A_A_Pcurr : INT ;
   RFS_A_B_Pcurr : INT ;
   RFS_A_C_Pcurr : INT ;
   RFS_A_RT : REAL ;
   RFS_A_FltNo : INT ;
   T6_XPF_A1_ToHMI : WORD ;
   T6_XPF_A1_A_Pcurr : INT ;
   T6_XPF_A1_B_Pcurr : INT ;
   T6_XPF_A1_C_Pcurr : INT ;
   T6_XPF_A1_RT : REAL ;
   T6_XPF_A1_FltNo : INT ;
   T7_XPF_A1_ToHMI : WORD ;
   T7_XPF_A1_A_Pcurr : INT ;
   T7_XPF_A1_B_Pcurr : INT ;
   T7_XPF_A1_C_Pcurr : INT ;
   T7_XPF_A1_RT : REAL ;
   T7_XPF_A1_FltNo : INT ;
   K4_XK_A1_ToHMI : WORD ;
   K4_XK_A1_A_Pcurr : INT ;
   K4_XK_A1_B_Pcurr : INT ;
   K4_XK_A1_C_Pcurr : INT ;
   K4_XK_A1_RT : REAL ;
   K4_XK_A1_FltNo : INT ;
   K4_HPF_A1_ToHMI : WORD ;
   K4_HPF_A1_A_Pcurr : INT ;
   K4_HPF_A1_B_Pcurr : INT ;
   K4_HPF_A1_C_Pcurr : INT ;
   K4_HPF_A1_RT : REAL ;
   K4_HPF_A1_FltNo : INT ;
   YL_IMCC_FJ_1_ToHMI : WORD ;
   YL_IMCC_FJ_1_Pcurr : INT ;
   YL_IMCC_FJ_1_RunTime : REAL ;
   YL_IMCC_FJ_1_FltNo : INT ;
   YL_IMCC_FJ_2_ToHMI : WORD ;
   YL_IMCC_FJ_2_Pcurr : INT ;
   YL_IMCC_FJ_2_RunTime : REAL ;
   YL_IMCC_FJ_2_FltNo : INT ;
   YL_IMCC_FJ_3_ToHMI : WORD ;
   YL_IMCC_FJ_3_Pcurr : INT ;
   YL_IMCC_FJ_3_RunTime : REAL ;
   YL_IMCC_FJ_3_FltNo : INT ;
   YL_IMCC_FJ_4_ToHMI : WORD ;
   YL_IMCC_FJ_4_Pcurr : INT ;
   YL_IMCC_FJ_4_RunTime : REAL ;
   YL_IMCC_FJ_4_FltNo : INT ;
   YL_IMCC_FJ_5_ToHMI : WORD ;
   YL_IMCC_FJ_5_Pcurr : INT ;
   YL_IMCC_FJ_5_RunTime : REAL ;
   YL_IMCC_FJ_5_FltNo : INT ;
   RFM_ToHMI : WORD ;
   JH_YC_A_ToHMI : WORD ;
   E420_01_N_ToHMI : WORD ;
   E420_05_K_ToHMI : WORD ;
   E420_06_K_ToHMI : WORD ;
   E420_07_K_ToHMI : WORD ;
   YL_FT1_ToHMI : WORD ;
   H420_01_N_ToHMI : WORD ;
   H420_01_N_FLOOR : WORD ;
   EPS21_ToHMI1 : WORD ;
   EPS21_ToHMI : ARRAY  [0 .. 15 ] OF INT  := 0;
   EPS11_ToHMI1 : WORD ;
   EPS11_ToHMI : ARRAY  [0 .. 15 ] OF INT ;
   WLE_1_ToHMI : WORD ;
   WLE_2_ToHMI : WORD ;
   WLE_3_ToHMI : WORD ;
   WLE_4_ToHMI : WORD ;
   IMCC_Com_A : WORD ;
  END_STRUCT ;	
BEGIN
END_DATA_BLOCK

DATA_BLOCK DB 6005
VERSION : 0.0
"HF3_Mode_Explode_FB3005"
BEGIN
END_DATA_BLOCK

DATA_BLOCK "HF3_DP_Statu_ToHMI"	// DB 6009
VERSION : 0.1
  STRUCT
   DP3_STATUS : ARRAY  [0 .. 15 ] OF //Status of module DPslave3 true means bad
   BOOL  := FALSE;
   DP4_STATUS : ARRAY  [0 .. 15 ] OF //Status of module DPslave4
   BOOL  := FALSE;
   DP5_STATUS : ARRAY  [0 .. 15 ] OF //Status of module DPslave5
   BOOL  := FALSE;
   DP6_STATUS : ARRAY  [0 .. 15 ] OF //Status of module DPslave6
   BOOL  := FALSE;
   DP7_STATUS : ARRAY  [0 .. 15 ] OF //Status of module DPslave7
   BOOL  := FALSE;
   DP8_STATUS : ARRAY  [0 .. 15 ] OF //Status of module DPslave8
   BOOL  := FALSE;
   DP9_STATUS : ARRAY  [0 .. 15 ] OF //Status of module DPslave9
   BOOL  := FALSE;
   DP10_STATUS : ARRAY  [0 .. 15 ] OF //Status of module DPslave10
   BOOL  := FALSE;
   DP11_STATUS : ARRAY  [0 .. 15 ] OF //Status of module DPslave11
   BOOL  := FALSE;
   DP12_STATUS : ARRAY  [0 .. 15 ] OF //Status of module DPslave12
   BOOL  := FALSE;
   DP13_STATUS : ARRAY  [0 .. 15 ] OF //Status of module DPslave13
   BOOL  := FALSE;
   DP14_STATUS : ARRAY  [0 .. 15 ] OF //Status of module DPslave14
   BOOL  := FALSE;
   DP15_STATUS : ARRAY  [0 .. 15 ] OF //Status of module DPslave15
   BOOL  := FALSE;
   DP16_STATUS : ARRAY  [0 .. 15 ] OF //Status of module DPslave16
   BOOL  := FALSE;
   DP17_STATUS : ARRAY  [0 .. 15 ] OF //Status of module DPslave17
   BOOL  := FALSE;
   DP18_STATUS : ARRAY  [0 .. 15 ] OF //Status of module DPslave18
   BOOL  := FALSE;
   DP19_STATUS : ARRAY  [0 .. 15 ] OF //Status of module DPslave19
   BOOL  := FALSE;
   DP20_STATUS : ARRAY  [0 .. 15 ] OF //Status of module DPslave20
   BOOL  := FALSE;
   DP21_STATUS : ARRAY  [0 .. 15 ] OF //Status of module DPslave21
   BOOL  := FALSE;
   DP22_STATUS : ARRAY  [0 .. 15 ] OF //Status of module DPslave22
   BOOL  := FALSE;
   DP23_STATUS : ARRAY  [0 .. 15 ] OF //Status of module DPslave23
   BOOL  := FALSE;
   DP24_STATUS : ARRAY  [0 .. 15 ] OF //Status of module DPslave24
   BOOL  := FALSE;
   DP25_STATUS : ARRAY  [0 .. 15 ] OF //Status of module DPslave25
   BOOL  := FALSE;
   DP26_STATUS : ARRAY  [0 .. 15 ] OF //Status of module DPslave26
   BOOL  := FALSE;
   DP27_STATUS : ARRAY  [0 .. 15 ] OF //Status of module DPslave27
   BOOL  := FALSE;
   DP28_STATUS : ARRAY  [0 .. 15 ] OF //Status of module DPslave28
   BOOL  := FALSE;
   DP29_STATUS : ARRAY  [0 .. 15 ] OF //Status of module DPslave29
   BOOL  := FALSE;
   DP30_STATUS : ARRAY  [0 .. 15 ] OF //Status of module DPslave30
   BOOL  := FALSE;
   DP31_STATUS : ARRAY  [0 .. 15 ] OF //Status of module DPslave31
   BOOL  := FALSE;
   DP32_STATUS : ARRAY  [0 .. 15 ] OF //Status of module DPslave32
   BOOL  := FALSE;
   DP33_STATUS : ARRAY  [0 .. 15 ] OF //Status of module DPslave33
   BOOL  := FALSE;
   DP34_STATUS : ARRAY  [0 .. 15 ] OF //Status of module DPslave34
   BOOL  := FALSE;
   DP35_STATUS : ARRAY  [0 .. 15 ] OF //Status of module DPslave35
   BOOL  := FALSE;
   DP36_STATUS : ARRAY  [0 .. 15 ] OF //Status of module DPslave36
   BOOL  := FALSE;
   DP37_STATUS : ARRAY  [0 .. 15 ] OF //Status of module DPslave37
   BOOL  := FALSE;
   DP38_STATUS : ARRAY  [0 .. 15 ] OF //Status of module DPslave38
   BOOL  := FALSE;
   DP39_STATUS : ARRAY  [0 .. 15 ] OF //Status of module DPslave39
   BOOL  := FALSE;
   DP40_STATUS : ARRAY  [0 .. 15 ] OF //Status of module DPslave40
   BOOL  := FALSE;
   DP41_STATUS : ARRAY  [0 .. 15 ] OF //Status of module DPslave41
   BOOL  := FALSE;
   DP42_STATUS : ARRAY  [0 .. 15 ] OF //Status of module DPslave42
   BOOL  := FALSE;
   DP43_STATUS : ARRAY  [0 .. 15 ] OF //Status of module DPslave43
   BOOL  := FALSE;
   DP44_STATUS : ARRAY  [0 .. 15 ] OF //Status of module DPslave44
   BOOL  := FALSE;
   DP45_STATUS : ARRAY  [0 .. 15 ] OF //Status of module DPslave45
   BOOL  := FALSE;
   DP46_STATUS : ARRAY  [0 .. 15 ] OF //Status of module DPslave46
   BOOL  := FALSE;
   DP47_STATUS : ARRAY  [0 .. 15 ] OF //Status of module DPslave47
   BOOL  := FALSE;
   DP48_STATUS : ARRAY  [0 .. 15 ] OF //Status of module DPslave48
   BOOL  := FALSE;
   DP49_STATUS : ARRAY  [0 .. 15 ] OF //Status of module DPslave49
   BOOL  := FALSE;
   DP50_STATUS : ARRAY  [0 .. 15 ] OF //Status of module DPslave50
   BOOL  := FALSE;
   DP51_STATUS : ARRAY  [0 .. 15 ] OF //Status of module DPslave51
   BOOL  := FALSE;
   DP52_STATUS : ARRAY  [0 .. 15 ] OF //Status of module DPslave52
   BOOL  := FALSE;
   DP3_Comm_Rack0 : WORD ;	//Status of communication of dp slave form rack0
   DP4_Comm_Rack0 : WORD ;	//Status of communication of dp slave form rack0
   DP5_Comm_Rack0 : WORD ;	//Status of communication of dp slave form rack0
   DP6_Comm_Rack0 : WORD ;	//Status of communication of dp slave form rack0
   DP7_Comm_Rack0 : WORD ;	//Status of communication of dp slave form rack0
   DP8_Comm_Rack0 : WORD ;	//Status of communication of dp slave form rack0
   DP9_Comm_Rack0 : WORD ;	//Status of communication of dp slave form rack0
   DP10_Comm_Rack0 : WORD ;	//Status of communication of dp slave form rack0
   DP11_Comm_Rack0 : WORD ;	//Status of communication of dp slave form rack0
   DP12_Comm_Rack0 : WORD ;	//Status of communication of dp slave form rack0
   DP13_Comm_Rack0 : WORD ;	//Status of communication of dp slave form rack0
   DP14_Comm_Rack0 : WORD ;	//Status of communication of dp slave form rack0
   DP15_Comm_Rack0 : WORD ;	//Status of communication of dp slave form rack0
   DP16_Comm_Rack0 : WORD ;	//Status of communication of dp slave form rack0
   DP17_Comm_Rack0 : WORD ;	//Status of communication of dp slave form rack0
   DP18_Comm_Rack0 : WORD ;	//Status of communication of dp slave form rack0
   DP19_Comm_Rack0 : WORD ;	//Status of communication of dp slave form rack0
   DP20_Comm_Rack0 : WORD ;	//Status of communication of dp slave form rack0
   DP21_Comm_Rack0 : WORD ;	//Status of communication of dp slave form rack0
   DP22_Comm_Rack0 : WORD ;	//Status of communication of dp slave form rack0
   DP23_Comm_Rack0 : WORD ;	//Status of communication of dp slave form rack0
   DP24_Comm_Rack0 : WORD ;	//Status of communication of dp slave form rack0
   DP25_Comm_Rack0 : WORD ;	//Status of communication of dp slave form rack0
   DP26_Comm_Rack0 : WORD ;	//Status of communication of dp slave form rack0
   DP27_Comm_Rack0 : WORD ;	//Status of communication of dp slave form rack0
   DP28_Comm_Rack0 : WORD ;	//Status of communication of dp slave form rack0
   DP29_Comm_Rack0 : WORD ;	//Status of communication of dp slave form rack0
   DP30_Comm_Rack0 : WORD ;	//Status of communication of dp slave form rack0
   DP31_Comm_Rack0 : WORD ;	//Status of communication of dp slave form rack0
   DP32_Comm_Rack0 : WORD ;	//Status of communication of dp slave form rack0
   DP33_Comm_Rack0 : WORD ;	//Status of communication of dp slave form rack0
   DP34_Comm_Rack0 : WORD ;	//Status of communication of dp slave form rack0
   DP35_Comm_Rack0 : WORD ;	//Status of communication of dp slave form rack0
   DP36_Comm_Rack0 : WORD ;	//Status of communication of dp slave form rack0
   DP37_Comm_Rack0 : WORD ;	//Status of communication of dp slave form rack0
   DP38_Comm_Rack0 : WORD ;	//Status of communication of dp slave form rack0
   DP39_Comm_Rack0 : WORD ;	//Status of communication of dp slave form rack0
   DP40_Comm_Rack0 : WORD ;	//Status of communication of dp slave form rack0
   DP41_Comm_Rack0 : WORD ;	//Status of communication of dp slave form rack0
   DP42_Comm_Rack0 : WORD ;	//Status of communication of dp slave form rack0
   DP43_Comm_Rack0 : WORD ;	//Status of communication of dp slave form rack0
   DP44_Comm_Rack0 : WORD ;	//Status of communication of dp slave form rack0
   DP45_Comm_Rack0 : WORD ;	//Status of communication of dp slave form rack0
   DP46_Comm_Rack0 : WORD ;	//Status of communication of dp slave form rack0
   DP47_Comm_Rack0 : WORD ;	//Status of communication of dp slave form rack0
   DP48_Comm_Rack0 : WORD ;	//Status of communication of dp slave form rack0
   DP49_Comm_Rack0 : WORD ;	//Status of communication of dp slave form rack0
   DP50_Comm_Rack0 : WORD ;	//Status of communication of dp slave form rack0
   DP51_Comm_Rack0 : WORD ;	//Status of communication of dp slave form rack0
   DP52_Comm_Rack0 : WORD ;	//Status of communication of dp slave form rack0
   DP3_Comm_Rack1 : WORD ;	//Status of communication of dp slave form rack1
   DP4_Comm_Rack1 : WORD ;	//Status of communication of dp slave form rack1
   DP5_Comm_Rack1 : WORD ;	//Status of communication of dp slave form rack1
   DP6_Comm_Rack1 : WORD ;	//Status of communication of dp slave form rack1
   DP7_Comm_Rack1 : WORD ;	//Status of communication of dp slave form rack1
   DP8_Comm_Rack1 : WORD ;	//Status of communication of dp slave form rack1
   DP9_Comm_Rack1 : WORD ;	//Status of communication of dp slave form rack1
   DP10_Comm_Rack1 : WORD ;	//Status of communication of dp slave form rack1
   DP11_Comm_Rack1 : WORD ;	//Status of communication of dp slave form rack1
   DP12_Comm_Rack1 : WORD ;	//Status of communication of dp slave form rack1
   DP13_Comm_Rack1 : WORD ;	//Status of communication of dp slave form rack1
   DP14_Comm_Rack1 : WORD ;	//Status of communication of dp slave form rack0
   DP15_Comm_Rack1 : WORD ;	//Status of communication of dp slave form rack0
   DP16_Comm_Rack1 : WORD ;	//Status of communication of dp slave form rack0
   DP17_Comm_Rack1 : WORD ;	//Status of communication of dp slave form rack0
   DP18_Comm_Rack1 : WORD ;	//Status of communication of dp slave form rack0
   DP19_Comm_Rack1 : WORD ;	//Status of communication of dp slave form rack0
   DP20_Comm_Rack1 : WORD ;	//Status of communication of dp slave form rack0
   DP21_Comm_Rack1 : WORD ;	//Status of communication of dp slave form rack0
   DP22_Comm_Rack1 : WORD ;	//Status of communication of dp slave form rack0
   DP23_Comm_Rack1 : WORD ;	//Status of communication of dp slave form rack0
   DP24_Comm_Rack1 : WORD ;	//Status of communication of dp slave form rack0
   DP25_Comm_Rack1 : WORD ;	//Status of communication of dp slave form rack0
   DP26_Comm_Rack1 : WORD ;	//Status of communication of dp slave form rack0
   DP27_Comm_Rack1 : WORD ;	//Status of communication of dp slave form rack0
   DP28_Comm_Rack1 : WORD ;	//Status of communication of dp slave form rack0
   DP29_Comm_Rack1 : WORD ;	//Status of communication of dp slave form rack0
   DP30_Comm_Rack1 : WORD ;	//Status of communication of dp slave form rack0
   DP31_Comm_Rack1 : WORD ;	//Status of communication of dp slave form rack0
   DP32_Comm_Rack1 : WORD ;	//Status of communication of dp slave form rack0
   DP33_Comm_Rack1 : WORD ;	//Status of communication of dp slave form rack0
   DP34_Comm_Rack1 : WORD ;	//Status of communication of dp slave form rack0
   DP35_Comm_Rack1 : WORD ;	//Status of communication of dp slave form rack0
   DP36_Comm_Rack1 : WORD ;	//Status of communication of dp slave form rack0
   DP37_Comm_Rack1 : WORD ;	//Status of communication of dp slave form rack0
   DP38_Comm_Rack1 : WORD ;	//Status of communication of dp slave form rack0
   DP39_Comm_Rack1 : WORD ;	//Status of communication of dp slave form rack0
   DP40_Comm_Rack1 : WORD ;	//Status of communication of dp slave form rack0
   DP41_Comm_Rack1 : WORD ;	//Status of communication of dp slave form rack0
   DP42_Comm_Rack1 : WORD ;	//Status of communication of dp slave form rack0
   DP43_Comm_Rack1 : WORD ;	//Status of communication of dp slave form rack0
   DP44_Comm_Rack1 : WORD ;	//Status of communication of dp slave form rack0
   DP45_Comm_Rack1 : WORD ;	//Status of communication of dp slave form rack0
   DP46_Comm_Rack1 : WORD ;	//Status of communication of dp slave form rack0
   DP47_Comm_Rack1 : WORD ;	//Status of communication of dp slave form rack0
   DP48_Comm_Rack1 : WORD ;	//Status of communication of dp slave form rack0
   DP49_Comm_Rack1 : WORD ;	//Status of communication of dp slave form rack0
   DP50_Comm_Rack1 : WORD ;	//Status of communication of dp slave form rack0
   DP51_Comm_Rack1 : WORD ;	//Status of communication of dp slave form rack0
   DP52_Comm_Rack1 : WORD ;	//Status of communication of dp slave form rack0
  END_STRUCT ;	
BEGIN
   DP4_STATUS[3] := TRUE;
   DP5_STATUS[3] := TRUE;
END_DATA_BLOCK

DATA_BLOCK "HF3_PLC_Statu_ToHMI"	// DB 6010
VERSION : 0.1
  STRUCT
   R0_Master : BOOL ;	//0号机架CPU是否为主CPU
   R0_RUN : BOOL ;	//0号机架CPU是否运行
   R0_PS_ERROR : BOOL ;	//0号机架CPU是否电池故障
   R0_EXTF_ERROR : BOOL ;	//0号机架CPU是否硬件故障
   R0_REDF_ERROR : BOOL ;	//0号机架CPU是否冗余故障
   DATA1 : BOOL ;
   DATA2 : BOOL ;
   DATA3 : BOOL ;
   R1_Master : BOOL ;	//1号机架CPU是否为主CPU
   R1_RUN : BOOL ;	//1号机架CPU是否运行
   R1_PS_ERROR : BOOL ;	//1号机架CPU是否电池故障
   R1_EXTF_ERROR : BOOL ;	//1号机架CPU是否硬件故障
   R1_REDF_ERROR : BOOL ;	//1号机架CPU是否冗余故障
  END_STRUCT ;	
BEGIN
END_DATA_BLOCK

DATA_BLOCK "给上位_状态"	// DB 6030
VERSION : 0.1
  STRUCT
   IMCC_Com_A : WORD ;
   KT_A1_ToHMI1 : WORD ;
   KT_A1_ToHMI2 : WORD ;
   KT_A1_VFRT : DWORD ;
   KT_A1_RPM : INT ;
   KT_A1_MotrCurr : INT ;
   KT_A1_AxleT : INT ;
   KT_A1_WindT : INT ;
   KT_A1_VFFB : INT ;
   KT_A1_RealTP : INT ;
   KT_A1_ECSum : DWORD ;
   KT_A1_FltNo : INT ;
   KT_A1_RT : REAL ;
   YL_KT_A1_1 : WORD ;
   YL_KT_A1_2 : WORD ;
   YL_KT_A1_3 : WORD ;
   IMCC_Com_B : WORD ;
   HPF_A1_ToHMI1 : WORD ;
   HPF_A1_ToHMI2 : WORD ;
   HPF_A1_VFFB : INT ;
   HPF_A1_A_Pcurr : INT ;
   HPF_A1_B_Pcurr : INT ;
   HPF_A1_C_Pcurr : INT ;
   HPF_A1_A_Pvolt : INT ;
   HPF_A1_B_Pvolt : INT ;
   HPF_A1_C_Pvolt : INT ;
   HPF_A1_RT : REAL ;
   HPF_A1_FltNo : INT ;
   YL_HPF_A1_1 : WORD ;
   YL_HPF_A1_2 : WORD ;
   YL_HPF_A1_3 : WORD ;
   YL_HPF_A1_4 : WORD ;
   DTS_A1_ToHMI : WORD ;
   DTS_A2_ToHMI : WORD ;
   DTS_A3_ToHMI : WORD ;
   DTS_A4_ToHMI : WORD ;
   DTS_A5_ToHMI : WORD ;
   DTS_A6_ToHMI : WORD ;
   DTS_A7_ToHMI : WORD ;
   DTS_A8_ToHMI : WORD ;
   DTS_A9_ToHMI : WORD ;
   DTS_A10_ToHMI : WORD ;
   YL_BigA_1 : WORD ;
   YL_BigA_2 : WORD ;
   UOF_A1_ToHMI1 : WORD ;
   UOF_A1_ToHMI2 : WORD ;
   UOF_A1_VFFB : INT ;
   UOF_A1_A_Pcurr : INT ;
   UOF_A1_B_Pcurr : INT ;
   UOF_A1_C_Pcurr : INT ;
   UOF_A1_A_Pvolt : INT ;
   UOF_A1_B_Pvolt : INT ;
   UOF_A1_C_Pvolt : INT ;
   UOF_A1_FAxleT : INT ;
   UOF_A1_RAxleT : INT ;
   UOF_A1_A_WindT : INT ;
   UOF_A1_B_WindT : INT ;
   UOF_A1_C_WindT : INT ;
   UOF_A1_X_Vibr : INT ;
   UOF_A1_Y_Vibr : INT ;
   UOF_A1_RT : REAL ;
   UOF_A1_FltNo : INT ;
   YL_UOF_A1_1 : WORD ;
   YL_UOF_A1_2 : WORD ;
   YL_UOF_A1_3 : WORD ;
   YL_UOF_A1_4 : WORD ;
   TVF_A1_ToHMI1 : WORD ;
   TVF_A1_ToHMI2 : WORD ;
   TVF_A1_A_Pcurr : INT ;
   TVF_A1_B_Pcurr : INT ;
   TVF_A1_C_Pcurr : INT ;
   TVF_A1_A_Pvolt : INT ;
   TVF_A1_B_Pvolt : INT ;
   TVF_A1_C_Pvolt : INT ;
   TVF_A1_FAxleT : INT ;
   TVF_A1_RAxleT : INT ;
   TVF_A1_A_WindT : INT ;
   TVF_A1_B_WindT : INT ;
   TVF_A1_C_WindT : INT ;
   TVF_A1_X_Vibr : INT ;
   TVF_A1_Y_Vibr : INT ;
   TVF_A1_RT : REAL ;
   TVF_A1_FltNo : INT ;
   YL_TVF_A1_1 : WORD ;
   YL_TVF_A1_2 : WORD ;
   YL_TVF_A1_3 : WORD ;
   YL_TVF_A1_4 : WORD ;
   TVF_A2_ToHMI1 : WORD ;
   TVF_A2_ToHMI2 : WORD ;
   TVF_A2_A_Pcurr : INT ;
   TVF_A2_B_Pcurr : INT ;
   TVF_A2_C_Pcurr : INT ;
   TVF_A2_A_Pvolt : INT ;
   TVF_A2_B_Pvolt : INT ;
   TVF_A2_C_Pvolt : INT ;
   TVF_A2_FAxleT : INT ;
   TVF_A2_RAxleT : INT ;
   TVF_A2_A_WindT : INT ;
   TVF_A2_B_WindT : INT ;
   TVF_A2_C_WindT : INT ;
   TVF_A2_X_Vibr : INT ;
   TVF_A2_Y_Vibr : INT ;
   TVF_A2_RT : REAL ;
   TVF_A2_FltNo : INT ;
   YL_TVF_A2_1 : WORD ;
   YL_TVF_A2_2 : WORD ;
   YL_TVF_A2_3 : WORD ;
   YL_TVF_A2_4 : WORD ;
   DM_A1_ToHMI : WORD ;
   DM_A2_ToHMI : WORD ;
   DM_A3_ToHMI : WORD ;
   DM_A4_ToHMI : WORD ;
   DM_A5_ToHMI : WORD ;
   DM_A6_ToHMI : WORD ;
   DM_A7_ToHMI : WORD ;
   DM_A8_ToHMI : WORD ;
   DM_A9_ToHMI : WORD ;
   DM_A10_ToHMI : WORD ;
   UOF_DT_A1_ToHMI : WORD ;
   UOF_DT_A2_ToHMI : WORD ;
   UOF_DT_A3_ToHMI : WORD ;
   UOF_DT_A4_ToHMI : WORD ;
   UOF_DT_A5_ToHMI : WORD ;
   UOF_DT_A6_ToHMI : WORD ;
   YL_TubA_1 : WORD ;
   YL_TubA_2 : WORD ;
   K1_XK_A1_ToHMI : WORD ;
   K1_XK_A1_A_Pcurr : INT ;
   K1_XK_A1_B_Pcurr : INT ;
   K1_XK_A1_C_Pcurr : INT ;
   K1_XK_A1_RT : REAL ;
   K1_XK_A1_FltNo : INT ;
   K1_HPF_A1_ToHMI : WORD ;
   K1_HPF_A1_A_Pcurr : INT ;
   K1_HPF_A1_B_Pcurr : INT ;
   K1_HPF_A1_C_Pcurr : INT ;
   K1_HPF_A1_RT : REAL ;
   K1_HPF_A1_FltNo : INT ;
   K1_DTS_A1_ToHMI : WORD ;
   K1_DTS_A2_ToHMI : WORD ;
   K1_DTS_A3_ToHMI : WORD ;
   K2_XK_A1_ToHMI : WORD ;
   K2_XK_A1_A_Pcurr : INT ;
   K2_XK_A1_B_Pcurr : INT ;
   K2_XK_A1_C_Pcurr : INT ;
   K2_XK_A1_RT : REAL ;
   K2_XK_A1_FltNo : INT ;
   K2_HPF_A1_ToHMI : WORD ;
   K2_HPF_A1_A_Pcurr : INT ;
   K2_HPF_A1_B_Pcurr : INT ;
   K2_HPF_A1_C_Pcurr : INT ;
   K2_HPF_A1_RT : REAL ;
   K2_HPF_A1_FltNo : INT ;
   K2_DTS_A1_ToHMI : WORD ;
   K2_DTS_A2_ToHMI : WORD ;
   K2_DTS_A3_ToHMI : WORD ;
   K3_XK_A1_ToHMI : WORD ;
   K3_XK_A1_A_Pcurr : INT ;
   K3_XK_A1_B_Pcurr : INT ;
   K3_XK_A1_C_Pcurr : INT ;
   K3_XK_A1_RT : REAL ;
   K3_XK_A1_FltNo : INT ;
   K3_HPF_A1_ToHMI : WORD ;
   K3_HPF_A1_A_Pcurr : INT ;
   K3_HPF_A1_B_Pcurr : INT ;
   K3_HPF_A1_C_Pcurr : INT ;
   K3_HPF_A1_RT : REAL ;
   K3_HPF_A1_FltNo : INT ;
   K3_DTS_A1_ToHMI : WORD ;
   K3_DTS_A2_ToHMI : WORD ;
   K3_DTS_A3_ToHMI : WORD ;
   K4_XK_A1_ToHMI : WORD ;
   K4_XK_A1_A_Pcurr : INT ;
   K4_XK_A1_B_Pcurr : INT ;
   K4_XK_A1_C_Pcurr : INT ;
   K4_XK_A1_RT : REAL ;
   K4_XK_A1_FltNo : INT ;
   K4_HPF_A1_ToHMI : WORD ;
   K4_HPF_A1_A_Pcurr : INT ;
   K4_HPF_A1_B_Pcurr : INT ;
   K4_HPF_A1_C_Pcurr : INT ;
   K4_HPF_A1_RT : REAL ;
   K4_HPF_A1_FltNo : INT ;
   K4_DTS_A1_ToHMI : WORD ;
   K4_DTS_A2_ToHMI : WORD ;
   K4_DTS_A3_ToHMI : WORD ;
   K5_XK_A1_ToHMI : WORD ;
   K5_XK_A1_A_Pcurr : INT ;
   K5_XK_A1_B_Pcurr : INT ;
   K5_XK_A1_C_Pcurr : INT ;
   K5_XK_A1_RT : REAL ;
   K5_XK_A1_FltNo : INT ;
   K5_HPF_A1_ToHMI : WORD ;
   K5_HPF_A1_A_Pcurr : INT ;
   K5_HPF_A1_B_Pcurr : INT ;
   K5_HPF_A1_C_Pcurr : INT ;
   K5_HPF_A1_RT : REAL ;
   K5_HPF_A1_FltNo : INT ;
   K5_DTS_A1_ToHMI : WORD ;
   K5_DTS_A2_ToHMI : WORD ;
   K5_DTS_A3_ToHMI : WORD ;
   K6_XK_A1_ToHMI : WORD ;
   K6_XK_A1_A_Pcurr : INT ;
   K6_XK_A1_B_Pcurr : INT ;
   K6_XK_A1_C_Pcurr : INT ;
   K6_XK_A1_RT : REAL ;
   K6_XK_A1_FltNo : INT ;
   K6_HPF_A1_ToHMI : WORD ;
   K6_HPF_A1_A_Pcurr : INT ;
   K6_HPF_A1_B_Pcurr : INT ;
   K6_HPF_A1_C_Pcurr : INT ;
   K6_HPF_A1_RT : REAL ;
   K6_HPF_A1_FltNo : INT ;
   K6_DTS_A1_ToHMI : WORD ;
   K6_DTS_A2_ToHMI : WORD ;
   K6_DTS_A3_ToHMI : WORD ;
   K7_XK_A1_ToHMI : WORD ;
   K7_XK_A1_A_Pcurr : INT ;
   K7_XK_A1_B_Pcurr : INT ;
   K7_XK_A1_C_Pcurr : INT ;
   K7_XK_A1_RT : REAL ;
   K7_XK_A1_FltNo : INT ;
   K7_HPF_A1_ToHMI : WORD ;
   K7_HPF_A1_A_Pcurr : INT ;
   K7_HPF_A1_B_Pcurr : INT ;
   K7_HPF_A1_C_Pcurr : INT ;
   K7_HPF_A1_RT : REAL ;
   K7_HPF_A1_FltNo : INT ;
   K7_DTS_A1_ToHMI : WORD ;
   K7_DTS_A2_ToHMI : WORD ;
   K7_DTS_A3_ToHMI : WORD ;
   T1_XSF_A1_ToHMI : WORD ;
   T1_XSF_A1_A_Pcurr : INT ;
   T1_XSF_A1_B_Pcurr : INT ;
   T1_XSF_A1_C_Pcurr : INT ;
   T1_XSF_A1_RT : REAL ;
   T1_XSF_A1_FltNo : INT ;
   T1_XPF_A1_ToHMI : WORD ;
   T1_XPF_A1_A_Pcurr : INT ;
   T1_XPF_A1_B_Pcurr : INT ;
   T1_XPF_A1_C_Pcurr : INT ;
   T1_XPF_A1_RT : REAL ;
   T1_XPF_A1_FltNo : INT ;
   T1_D_A1_ToHMI : WORD ;
   T1_D_A2_ToHMI : WORD ;
   T2_XSF_A1_ToHMI : WORD ;
   T2_XSF_A1_A_Pcurr : INT ;
   T2_XSF_A1_B_Pcurr : INT ;
   T2_XSF_A1_C_Pcurr : INT ;
   T2_XSF_A1_RT : REAL ;
   T2_XSF_A1_FltNo : INT ;
   T2_XPF_A1_ToHMI : WORD ;
   T2_XPF_A1_A_Pcurr : INT ;
   T2_XPF_A1_B_Pcurr : INT ;
   T2_XPF_A1_C_Pcurr : INT ;
   T2_XPF_A1_RT : REAL ;
   T2_XPF_A1_FltNo : INT ;
   T2_D_A1_ToHMI : WORD ;
   T2_D_A2_ToHMI : WORD ;
   T3_XSF_A1_ToHMI : WORD ;
   T3_XSF_A1_A_Pcurr : INT ;
   T3_XSF_A1_B_Pcurr : INT ;
   T3_XSF_A1_C_Pcurr : INT ;
   T3_XSF_A1_RT : REAL ;
   T3_XSF_A1_FltNo : INT ;
   T3_XPF_A1_ToHMI : WORD ;
   T3_XPF_A1_A_Pcurr : INT ;
   T3_XPF_A1_B_Pcurr : INT ;
   T3_XPF_A1_C_Pcurr : INT ;
   T3_XPF_A1_RT : REAL ;
   T3_XPF_A1_FltNo : INT ;
   T3_D_A1_ToHMI : WORD ;
   T3_D_A2_ToHMI : WORD ;
   T4_XSF_A1_ToHMI : WORD ;
   T4_XSF_A1_A_Pcurr : INT ;
   T4_XSF_A1_B_Pcurr : INT ;
   T4_XSF_A1_C_Pcurr : INT ;
   T4_XSF_A1_RT : REAL ;
   T4_XSF_A1_FltNo : INT ;
   T4_XPF_A1_ToHMI : WORD ;
   T4_XPF_A1_A_Pcurr : INT ;
   T4_XPF_A1_B_Pcurr : INT ;
   T4_XPF_A1_C_Pcurr : INT ;
   T4_XPF_A1_RT : REAL ;
   T4_XPF_A1_FltNo : INT ;
   T4_D_A1_ToHMI : WORD ;
   T4_D_A2_ToHMI : WORD ;
   T5_XSF_A1_ToHMI : WORD ;
   T5_XSF_A1_A_Pcurr : INT ;
   T5_XSF_A1_B_Pcurr : INT ;
   T5_XSF_A1_C_Pcurr : INT ;
   T5_XSF_A1_RT : REAL ;
   T5_XSF_A1_FltNo : INT ;
   T5_XPF_A1_ToHMI : WORD ;
   T5_XPF_A1_A_Pcurr : INT ;
   T5_XPF_A1_B_Pcurr : INT ;
   T5_XPF_A1_C_Pcurr : INT ;
   T5_XPF_A1_RT : REAL ;
   T5_XPF_A1_FltNo : INT ;
   T5_D_A1_ToHMI : WORD ;
   T5_D_A2_ToHMI : WORD ;
   T6_XSF_A1_ToHMI : WORD ;
   T6_XSF_A1_A_Pcurr : INT ;
   T6_XSF_A1_B_Pcurr : INT ;
   T6_XSF_A1_C_Pcurr : INT ;
   T6_XSF_A1_RT : REAL ;
   T6_XSF_A1_FltNo : INT ;
   T6_XPF_A1_ToHMI : WORD ;
   T6_XPF_A1_A_Pcurr : INT ;
   T6_XPF_A1_B_Pcurr : INT ;
   T6_XPF_A1_C_Pcurr : INT ;
   T6_XPF_A1_RT : REAL ;
   T6_XPF_A1_FltNo : INT ;
   T6_D_A1_ToHMI : WORD ;
   T6_D_A2_ToHMI : WORD ;
   T7_XSF_A1_ToHMI : WORD ;
   T7_XSF_A1_A_Pcurr : INT ;
   T7_XSF_A1_B_Pcurr : INT ;
   T7_XSF_A1_C_Pcurr : INT ;
   T7_XSF_A1_RT : REAL ;
   T7_XSF_A1_FltNo : INT ;
   T7_XPF_A1_ToHMI : WORD ;
   T7_XPF_A1_A_Pcurr : INT ;
   T7_XPF_A1_B_Pcurr : INT ;
   T7_XPF_A1_C_Pcurr : INT ;
   T7_XPF_A1_RT : REAL ;
   T7_XPF_A1_FltNo : INT ;
   T7_D_A1_ToHMI : WORD ;
   T7_D_A2_ToHMI : WORD ;
   T8_XSF_A1_ToHMI : WORD ;
   T8_XSF_A1_A_Pcurr : INT ;
   T8_XSF_A1_B_Pcurr : INT ;
   T8_XSF_A1_C_Pcurr : INT ;
   T8_XSF_A1_RT : REAL ;
   T8_XSF_A1_FltNo : INT ;
   T8_XPF_A1_ToHMI : WORD ;
   T8_XPF_A1_A_Pcurr : INT ;
   T8_XPF_A1_B_Pcurr : INT ;
   T8_XPF_A1_C_Pcurr : INT ;
   T8_XPF_A1_RT : REAL ;
   T8_XPF_A1_FltNo : INT ;
   T8_XSF_A2_ToHMI : WORD ;
   T8_XSF_A2_A_Pcurr : INT ;
   T8_XSF_A2_B_Pcurr : INT ;
   T8_XSF_A2_C_Pcurr : INT ;
   T8_XSF_A2_RT : REAL ;
   T8_XSF_A2_FltNo : INT ;
   T8_XPF_A2_ToHMI : WORD ;
   T8_XPF_A2_A_Pcurr : INT ;
   T8_XPF_A2_B_Pcurr : INT ;
   T8_XPF_A2_C_Pcurr : INT ;
   T8_XPF_A2_RT : REAL ;
   T8_XPF_A2_FltNo : INT ;
   T8_D_A1_ToHMI : WORD ;
   T8_D_A2_ToHMI : WORD ;
   T8_D_A3_ToHMI : WORD ;
   T8_D_A4_ToHMI : WORD ;
   T8_D_A5_ToHMI : WORD ;
   T8_D_A6_ToHMI : WORD ;
   T8_D_A7_ToHMI : WORD ;
   T8_D_A8_ToHMI : WORD ;
   T8_D_A9_ToHMI : WORD ;
   T8_D_A10_ToHMI : WORD ;
   KT_B1_ToHMI1 : WORD ;
   KT_B1_ToHMI2 : WORD ;
   KT_B1_VFRT : DWORD ;
   KT_B1_RPM : INT ;
   KT_B1_MotrCurr : INT ;
   KT_B1_AxleT : INT ;
   KT_B1_WindT : INT ;
   KT_B1_VFFB : INT ;
   KT_B1_RealTP : INT ;
   KT_B1_ECSum : DWORD ;
   KT_B1_FltNo : INT ;
   KT_B1_RT : REAL ;
   YL_KT_B1_1 : WORD ;
   YL_KT_B1_2 : WORD ;
   YL_KT_B1_3 : WORD ;
   YL_KT_B1_4 : WORD ;
   HPF_B1_ToHMI1 : WORD ;
   HPF_B1_ToHMI2 : WORD ;
   HPF_B1_VFFB : INT ;
   HPF_B1_A_Pcurr : INT ;
   HPF_B1_B_Pcurr : INT ;
   HPF_B1_C_Pcurr : INT ;
   HPF_B1_A_Pvolt : INT ;
   HPF_B1_B_Pvolt : INT ;
   HPF_B1_C_Pvolt : INT ;
   HPF_B1_RT : REAL ;
   HPF_B1_FltNo : INT ;
   YL_HPF_B1_1 : WORD ;
   YL_HPF_B1_2 : WORD ;
   YL_HPF_B1_3 : WORD ;
   YL_HPF_B1_4 : WORD ;
   DTS_B1_ToHMI : WORD ;
   DTS_B2_ToHMI : WORD ;
   DTS_B3_ToHMI : WORD ;
   DTS_B4_ToHMI : WORD ;
   DTS_B5_ToHMI : WORD ;
   DTS_B6_ToHMI : WORD ;
   DTS_B7_ToHMI : WORD ;
   DTS_B8_ToHMI : WORD ;
   DTS_B9_ToHMI : WORD ;
   DTS_B10_ToHMI : WORD ;
   YL_BigB_1 : WORD ;
   YL_BigB_2 : WORD ;
   UOF_B1_ToHMI1 : WORD ;
   UOF_B1_ToHMI2 : WORD ;
   UOF_B1_VFFB : INT ;
   UOF_B1_A_Pcurr : INT ;
   UOF_B1_B_Pcurr : INT ;
   UOF_B1_C_Pcurr : INT ;
   UOF_B1_A_Pvolt : INT ;
   UOF_B1_B_Pvolt : INT ;
   UOF_B1_C_Pvolt : INT ;
   UOF_B1_FAxleT : INT ;
   UOF_B1_RAxleT : INT ;
   UOF_B1_A_WindT : INT ;
   UOF_B1_B_WindT : INT ;
   UOF_B1_C_WindT : INT ;
   UOF_B1_X_Vibr : INT ;
   UOF_B1_Y_Vibr : INT ;
   UOF_B1_RT : REAL ;
   UOF_B1_FltNo : INT ;
   YL_UOF_B1_1 : WORD ;
   YL_UOF_B1_2 : WORD ;
   YL_UOF_B1_3 : WORD ;
   YL_UOF_B1_4 : WORD ;
   TVF_B1_ToHMI1 : WORD ;
   TVF_B1_ToHMI2 : WORD ;
   TVF_B1_A_Pcurr : INT ;
   TVF_B1_B_Pcurr : INT ;
   TVF_B1_C_Pcurr : INT ;
   TVF_B1_A_Pvolt : INT ;
   TVF_B1_B_Pvolt : INT ;
   TVF_B1_C_Pvolt : INT ;
   TVF_B1_FAxleT : INT ;
   TVF_B1_RAxleT : INT ;
   TVF_B1_A_WindT : INT ;
   TVF_B1_B_WindT : INT ;
   TVF_B1_C_WindT : INT ;
   TVF_B1_X_Vibr : INT ;
   TVF_B1_Y_Vibr : INT ;
   TVF_B1_RT : REAL ;
   TVF_B1_FltNo : INT ;
   YL_TVF_B1_1 : WORD ;
   YL_TVF_B1_2 : WORD ;
   YL_TVF_B1_3 : WORD ;
   YL_TVF_B1_4 : WORD ;
   TVF_B2_ToHMI1 : WORD ;
   TVF_B2_ToHMI2 : WORD ;
   TVF_B2_A_Pcurr : INT ;
   TVF_B2_B_Pcurr : INT ;
   TVF_B2_C_Pcurr : INT ;
   TVF_B2_A_Pvolt : INT ;
   TVF_B2_B_Pvolt : INT ;
   TVF_B2_C_Pvolt : INT ;
   TVF_B2_FAxleT : INT ;
   TVF_B2_RAxleT : INT ;
   TVF_B2_A_WindT : INT ;
   TVF_B2_B_WindT : INT ;
   TVF_B2_C_WindT : INT ;
   TVF_B2_X_Vibr : INT ;
   TVF_B2_Y_Vibr : INT ;
   TVF_B2_RT : REAL ;
   TVF_B2_FltNo : INT ;
   YL_TVF_B2_1 : WORD ;
   YL_TVF_B2_2 : WORD ;
   YL_TVF_B2_3 : WORD ;
   YL_TVF_B2_4 : WORD ;
   DM_B1_ToHMI : WORD ;
   DM_B2_ToHMI : WORD ;
   DM_B3_ToHMI : WORD ;
   DM_B4_ToHMI : WORD ;
   DM_B5_ToHMI : WORD ;
   DM_B6_ToHMI : WORD ;
   DM_B7_ToHMI : WORD ;
   DM_B8_ToHMI : WORD ;
   DM_B9_ToHMI : WORD ;
   DM_B10_ToHMI : WORD ;
   UOF_DT_B1_ToHMI : WORD ;
   UOF_DT_B2_ToHMI : WORD ;
   UOF_DT_B3_ToHMI : WORD ;
   UOF_DT_B4_ToHMI : WORD ;
   UOF_DT_B5_ToHMI : WORD ;
   UOF_DT_B6_ToHMI : WORD ;
   YL_TubB_1 : WORD ;
   YL_TubB_2 : WORD ;
   K1_XK_B1_ToHMI : WORD ;
   K1_XK_B1_A_Pcurr : INT ;
   K1_XK_B1_B_Pcurr : INT ;
   K1_XK_B1_C_Pcurr : INT ;
   K1_XK_B1_RT : REAL ;
   K1_XK_B1_FltNo : INT ;
   K1_HPF_B1_ToHMI : WORD ;
   K1_HPF_B1_A_Pcurr : INT ;
   K1_HPF_B1_B_Pcurr : INT ;
   K1_HPF_B1_C_Pcurr : INT ;
   K1_HPF_B1_RT : REAL ;
   K1_HPF_B1_FltNo : INT ;
   K1_DTS_B1_ToHMI : WORD ;
   K1_DTS_B2_ToHMI : WORD ;
   K1_DTS_B3_ToHMI : WORD ;
   K2_XK_B1_ToHMI : WORD ;
   K2_XK_B1_A_Pcurr : INT ;
   K2_XK_B1_B_Pcurr : INT ;
   K2_XK_B1_C_Pcurr : INT ;
   K2_XK_B1_RT : REAL ;
   K2_XK_B1_FltNo : INT ;
   K2_HPF_B1_ToHMI : WORD ;
   K2_HPF_B1_A_Pcurr : INT ;
   K2_HPF_B1_B_Pcurr : INT ;
   K2_HPF_B1_C_Pcurr : INT ;
   K2_HPF_B1_RT : REAL ;
   K2_HPF_B1_FltNo : INT ;
   K2_DTS_B1_ToHMI : WORD ;
   K2_DTS_B2_ToHMI : WORD ;
   K2_DTS_B3_ToHMI : WORD ;
   K3_XK_B1_ToHMI : WORD ;
   K3_XK_B1_A_Pcurr : INT ;
   K3_XK_B1_B_Pcurr : INT ;
   K3_XK_B1_C_Pcurr : INT ;
   K3_XK_B1_RT : REAL ;
   K3_XK_B1_FltNo : INT ;
   K3_HPF_B1_ToHMI : WORD ;
   K3_HPF_B1_A_Pcurr : INT ;
   K3_HPF_B1_B_Pcurr : INT ;
   K3_HPF_B1_C_Pcurr : INT ;
   K3_HPF_B1_RT : REAL ;
   K3_HPF_B1_FltNo : INT ;
   K3_DTS_B1_ToHMI : WORD ;
   K3_DTS_B2_ToHMI : WORD ;
   K3_DTS_B3_ToHMI : WORD ;
   K4_XK_B1_ToHMI : WORD ;
   K4_XK_B1_A_Pcurr : INT ;
   K4_XK_B1_B_Pcurr : INT ;
   K4_XK_B1_C_Pcurr : INT ;
   K4_XK_B1_RT : REAL ;
   K4_XK_B1_FltNo : INT ;
   K4_HPF_B1_ToHMI : WORD ;
   K4_HPF_B1_A_Pcurr : INT ;
   K4_HPF_B1_B_Pcurr : INT ;
   K4_HPF_B1_C_Pcurr : INT ;
   K4_HPF_B1_RT : REAL ;
   K4_HPF_B1_FltNo : INT ;
   K4_DTS_B1_ToHMI : WORD ;
   K4_DTS_B2_ToHMI : WORD ;
   K4_DTS_B3_ToHMI : WORD ;
   K5_XK_B1_ToHMI : WORD ;
   K5_XK_B1_A_Pcurr : INT ;
   K5_XK_B1_B_Pcurr : INT ;
   K5_XK_B1_C_Pcurr : INT ;
   K5_XK_B1_RT : REAL ;
   K5_XK_B1_FltNo : INT ;
   K5_HPF_B1_ToHMI : WORD ;
   K5_HPF_B1_A_Pcurr : INT ;
   K5_HPF_B1_B_Pcurr : INT ;
   K5_HPF_B1_C_Pcurr : INT ;
   K5_HPF_B1_RT : REAL ;
   K5_HPF_B1_FltNo : INT ;
   K5_DTS_B1_ToHMI : WORD ;
   K5_DTS_B2_ToHMI : WORD ;
   K5_DTS_B3_ToHMI : WORD ;
   K6_XK_B1_ToHMI : WORD ;
   K6_XK_B1_A_Pcurr : INT ;
   K6_XK_B1_B_Pcurr : INT ;
   K6_XK_B1_C_Pcurr : INT ;
   K6_XK_B1_RT : REAL ;
   K6_XK_B1_FltNo : INT ;
   K6_HPF_B1_ToHMI : WORD ;
   K6_HPF_B1_A_Pcurr : INT ;
   K6_HPF_B1_B_Pcurr : INT ;
   K6_HPF_B1_C_Pcurr : INT ;
   K6_HPF_B1_RT : REAL ;
   K6_HPF_B1_FltNo : INT ;
   K6_DTS_B1_ToHMI : WORD ;
   K6_DTS_B2_ToHMI : WORD ;
   K6_DTS_B3_ToHMI : WORD ;
   K7_XK_B1_ToHMI : WORD ;
   K7_XK_B1_A_Pcurr : INT ;
   K7_XK_B1_B_Pcurr : INT ;
   K7_XK_B1_C_Pcurr : INT ;
   K7_XK_B1_RT : REAL ;
   K7_XK_B1_FltNo : INT ;
   K7_HPF_B1_ToHMI : WORD ;
   K7_HPF_B1_A_Pcurr : INT ;
   K7_HPF_B1_B_Pcurr : INT ;
   K7_HPF_B1_C_Pcurr : INT ;
   K7_HPF_B1_RT : REAL ;
   K7_HPF_B1_FltNo : INT ;
   K7_DTS_B1_ToHMI : WORD ;
   K7_DTS_B2_ToHMI : WORD ;
   K7_DTS_B3_ToHMI : WORD ;
   T1_XSF_B1_ToHMI : WORD ;
   T1_XSF_B1_A_Pcurr : INT ;
   T1_XSF_B1_B_Pcurr : INT ;
   T1_XSF_B1_C_Pcurr : INT ;
   T1_XSF_B1_RT : REAL ;
   T1_XSF_B1_FltNo : INT ;
   T1_XPF_B1_ToHMI : WORD ;
   T1_XPF_B1_A_Pcurr : INT ;
   T1_XPF_B1_B_Pcurr : INT ;
   T1_XPF_B1_C_Pcurr : INT ;
   T1_XPF_B1_RT : REAL ;
   T1_XPF_B1_FltNo : INT ;
   T1_D_B1_ToHMI : WORD ;
   T1_D_B2_ToHMI : WORD ;
   T2_XSF_B1_ToHMI : WORD ;
   T2_XSF_B1_A_Pcurr : INT ;
   T2_XSF_B1_B_Pcurr : INT ;
   T2_XSF_B1_C_Pcurr : INT ;
   T2_XSF_B1_RT : REAL ;
   T2_XSF_B1_FltNo : INT ;
   T2_XPF_B1_ToHMI : WORD ;
   T2_XPF_B1_A_Pcurr : INT ;
   T2_XPF_B1_B_Pcurr : INT ;
   T2_XPF_B1_C_Pcurr : INT ;
   T2_XPF_B1_RT : REAL ;
   T2_XPF_B1_FltNo : INT ;
   T2_D_B1_ToHMI : WORD ;
   T2_D_B2_ToHMI : WORD ;
   T3_XSF_B1_ToHMI : WORD ;
   T3_XSF_B1_A_Pcurr : INT ;
   T3_XSF_B1_B_Pcurr : INT ;
   T3_XSF_B1_C_Pcurr : INT ;
   T3_XSF_B1_RT : REAL ;
   T3_XSF_B1_FltNo : INT ;
   T3_XPF_B1_ToHMI : WORD ;
   T3_XPF_B1_A_Pcurr : INT ;
   T3_XPF_B1_B_Pcurr : INT ;
   T3_XPF_B1_C_Pcurr : INT ;
   T3_XPF_B1_RT : REAL ;
   T3_XPF_B1_FltNo : INT ;
   T3_D_B1_ToHMI : WORD ;
   T3_D_B2_ToHMI : WORD ;
   T4_XSF_B1_ToHMI : WORD ;
   T4_XSF_B1_A_Pcurr : INT ;
   T4_XSF_B1_B_Pcurr : INT ;
   T4_XSF_B1_C_Pcurr : INT ;
   T4_XSF_B1_RT : REAL ;
   T4_XSF_B1_FltNo : INT ;
   T4_XPF_B1_ToHMI : WORD ;
   T4_XPF_B1_A_Pcurr : INT ;
   T4_XPF_B1_B_Pcurr : INT ;
   T4_XPF_B1_C_Pcurr : INT ;
   T4_XPF_B1_RT : REAL ;
   T4_XPF_B1_FltNo : INT ;
   T4_D_B1_ToHMI : WORD ;
   T4_D_B2_ToHMI : WORD ;
   T5_XSF_B1_ToHMI : WORD ;
   T5_XSF_B1_A_Pcurr : INT ;
   T5_XSF_B1_B_Pcurr : INT ;
   T5_XSF_B1_C_Pcurr : INT ;
   T5_XSF_B1_RT : REAL ;
   T5_XSF_B1_FltNo : INT ;
   T5_XPF_B1_ToHMI : WORD ;
   T5_XPF_B1_A_Pcurr : INT ;
   T5_XPF_B1_B_Pcurr : INT ;
   T5_XPF_B1_C_Pcurr : INT ;
   T5_XPF_B1_RT : REAL ;
   T5_XPF_B1_FltNo : INT ;
   T5_D_B1_ToHMI : WORD ;
   T5_D_B2_ToHMI : WORD ;
   T6_XSF_B1_ToHMI : WORD ;
   T6_XSF_B1_A_Pcurr : INT ;
   T6_XSF_B1_B_Pcurr : INT ;
   T6_XSF_B1_C_Pcurr : INT ;
   T6_XSF_B1_RT : REAL ;
   T6_XSF_B1_FltNo : INT ;
   T6_XPF_B1_ToHMI : WORD ;
   T6_XPF_B1_A_Pcurr : INT ;
   T6_XPF_B1_B_Pcurr : INT ;
   T6_XPF_B1_C_Pcurr : INT ;
   T6_XPF_B1_RT : REAL ;
   T6_XPF_B1_FltNo : INT ;
   T6_D_B1_ToHMI : WORD ;
   T6_D_B2_ToHMI : WORD ;
   T7_XSF_B1_ToHMI : WORD ;
   T7_XSF_B1_A_Pcurr : INT ;
   T7_XSF_B1_B_Pcurr : INT ;
   T7_XSF_B1_C_Pcurr : INT ;
   T7_XSF_B1_RT : REAL ;
   T7_XSF_B1_FltNo : INT ;
   T7_XPF_B1_ToHMI : WORD ;
   T7_XPF_B1_A_Pcurr : INT ;
   T7_XPF_B1_B_Pcurr : INT ;
   T7_XPF_B1_C_Pcurr : INT ;
   T7_XPF_B1_RT : REAL ;
   T7_XPF_B1_FltNo : INT ;
   T7_D_B1_ToHMI : WORD ;
   T7_D_B2_ToHMI : WORD ;
   T8_XSF_B1_ToHMI : WORD ;
   T8_XSF_B1_A_Pcurr : INT ;
   T8_XSF_B1_B_Pcurr : INT ;
   T8_XSF_B1_C_Pcurr : INT ;
   T8_XSF_B1_RT : REAL ;
   T8_XSF_B1_FltNo : INT ;
   T8_XPF_B1_ToHMI : WORD ;
   T8_XPF_B1_A_Pcurr : INT ;
   T8_XPF_B1_B_Pcurr : INT ;
   T8_XPF_B1_C_Pcurr : INT ;
   T8_XPF_B1_RT : REAL ;
   T8_XPF_B1_FltNo : INT ;
   T8_XSF_B2_ToHMI : WORD ;
   T8_XSF_B2_A_Pcurr : INT ;
   T8_XSF_B2_B_Pcurr : INT ;
   T8_XSF_B2_C_Pcurr : INT ;
   T8_XSF_B2_RT : REAL ;
   T8_XSF_B2_FltNo : INT ;
   T8_XPF_B2_ToHMI : WORD ;
   T8_XPF_B2_A_Pcurr : INT ;
   T8_XPF_B2_B_Pcurr : INT ;
   T8_XPF_B2_C_Pcurr : INT ;
   T8_XPF_B2_RT : REAL ;
   T8_XPF_B2_FltNo : INT ;
   T8_D_B1_ToHMI : WORD ;
   T8_D_B2_ToHMI : WORD ;
   T8_D_B3_ToHMI : WORD ;
   T8_D_B4_ToHMI : WORD ;
   T8_D_B5_ToHMI : WORD ;
   T8_D_B6_ToHMI : WORD ;
   T8_D_B7_ToHMI : WORD ;
   T8_D_B8_ToHMI : WORD ;
   T8_D_B9_ToHMI : WORD ;
   T8_D_B10_ToHMI : WORD ;
   SB_1_ToHMI1 : WORD ;
   SB_1_ToHMI2 : WORD ;
   SB_1_Level : INT ;
   SB_1_RT : REAL ;
   SB_1_FltNo : INT ;
   SB_2_ToHMI1 : WORD ;
   SB_2_ToHMI2 : WORD ;
   SB_2_Level : INT ;
   SB_2_RT : REAL ;
   SB_2_FltNo : INT ;
   SB_3_ToHMI1 : WORD ;
   SB_3_ToHMI2 : WORD ;
   SB_3_Level : INT ;
   SB_3_RT : REAL ;
   SB_3_FltNo : INT ;
   SB_4_ToHMI1 : WORD ;
   SB_4_ToHMI2 : WORD ;
   SB_4_Level : INT ;
   SB_4_RT : REAL ;
   SB_4_FltNo : INT ;
   SB_5_ToHMI1 : WORD ;
   SB_5_ToHMI2 : WORD ;
   SB_5_Level : INT ;
   SB_5_RT : REAL ;
   SB_5_FltNo : INT ;
   SB_6_ToHMI1 : WORD ;
   SB_6_ToHMI2 : WORD ;
   SB_6_Level : INT ;
   SB_6_RT : REAL ;
   SB_6_FltNo : INT ;
   SB_7_ToHMI1 : WORD ;
   SB_7_ToHMI2 : WORD ;
   SB_7_Level : INT ;
   SB_7_RT : REAL ;
   SB_7_FltNo : INT ;
   SB_8_ToHMI1 : WORD ;
   SB_8_ToHMI2 : WORD ;
   SB_8_Level : INT ;
   SB_8_RT : REAL ;
   SB_8_FltNo : INT ;
   SB_9_ToHMI1 : WORD ;
   SB_9_ToHMI2 : WORD ;
   SB_9_Level : INT ;
   SB_9_RT : REAL ;
   SB_9_FltNo : INT ;
   SB_10_ToHMI1 : WORD ;
   SB_10_ToHMI2 : WORD ;
   SB_10_Level : INT ;
   SB_10_RT : REAL ;
   SB_10_FltNo : INT ;
   SB_11_ToHMI1 : WORD ;
   SB_11_ToHMI2 : WORD ;
   SB_11_Level : INT ;
   SB_11_RT : REAL ;
   SB_11_FltNo : INT ;
   SB_12_ToHMI1 : WORD ;
   SB_12_ToHMI2 : WORD ;
   SB_12_Level : INT ;
   SB_12_RT : REAL ;
   SB_12_FltNo : INT ;
   SB_13_ToHMI1 : WORD ;
   SB_13_ToHMI2 : WORD ;
   SB_13_Level : INT ;
   SB_13_RT : REAL ;
   SB_13_FltNo : INT ;
   SB_14_ToHMI1 : WORD ;
   SB_14_ToHMI2 : WORD ;
   SB_14_Level : INT ;
   SB_14_RT : REAL ;
   SB_14_FltNo : INT ;
   SB_15_ToHMI1 : WORD ;
   SB_15_ToHMI2 : WORD ;
   SB_15_Level : INT ;
   SB_15_RT : REAL ;
   SB_15_FltNo : INT ;
   SB_16_ToHMI1 : WORD ;
   SB_16_ToHMI2 : WORD ;
   SB_16_Level : INT ;
   SB_16_RT : REAL ;
   SB_16_FltNo : INT ;
   SB_17_ToHMI1 : WORD ;
   SB_17_ToHMI2 : WORD ;
   SB_17_Level : INT ;
   SB_17_RT : REAL ;
   SB_17_FltNo : INT ;
   SB_18_ToHMI1 : WORD ;
   SB_18_ToHMI2 : WORD ;
   SB_18_Level : INT ;
   SB_18_RT : REAL ;
   SB_18_FltNo : INT ;
   PSB_1_ToHMI : WORD ;
   PSB_1_Level : INT ;
   PSB_2_ToHMI : WORD ;
   PSB_2_Level : INT ;
   PSB_3_ToHMI : WORD ;
   PSB_3_Level : INT ;
   PSB_4_ToHMI : WORD ;
   PSB_4_Level : INT ;
   PSB_5_ToHMI : WORD ;
   PSB_5_Level : INT ;
   PSB_6_ToHMI : WORD ;
   PSB_6_Level : INT ;
   PSB_7_ToHMI : WORD ;
   PSB_7_Level : INT ;
   PSB_8_ToHMI : WORD ;
   PSB_8_Level : INT ;
   PSB_9_ToHMI : WORD ;
   PSB_9_Level : INT ;
   PSB_10_ToHMI : WORD ;
   PSB_10_Level : INT ;
   PSB_11_ToHMI : WORD ;
   PSB_11_Level : INT ;
   PSB_12_ToHMI : WORD ;
   PSB_12_Level : INT ;
   PSB_13_ToHMI : WORD ;
   PSB_13_Level : INT ;
   PSB_14_ToHMI : WORD ;
   PSB_14_Level : INT ;
   PSB_15_ToHMI : WORD ;
   PSB_15_Level : INT ;
   WSB_1_ToHMI : WORD ;
   WSB_1_Level : INT ;
   FT_1_ToHMI : WORD ;
   FT_2_ToHMI : WORD ;
   FT_3_ToHMI : WORD ;
   FT_4_ToHMI : WORD ;
   FT_5_ToHMI : WORD ;
   FT_6_ToHMI : WORD ;
   FT_7_ToHMI : WORD ;
   FT_8_ToHMI : WORD ;
   FT_9_ToHMI : WORD ;
   FT_10_ToHMI : WORD ;
   FT_11_ToHMI : WORD ;
   FT_12_ToHMI : WORD ;
   FT_13_ToHMI : WORD ;
   FT_14_ToHMI : WORD ;
   FT_15_ToHMI : WORD ;
   FT_16_ToHMI : WORD ;
   FT_17_ToHMI : WORD ;
   FT_18_ToHMI : WORD ;
   FT_19_ToHMI : WORD ;
   FT_20_ToHMI : WORD ;
   DT_1_ToHMI : WORD ;
   DT_1_Floor : WORD ;
   DT_2_ToHMI : WORD ;
   DT_2_Floor : WORD ;
   DT_3_ToHMI : WORD ;
   DT_3_Floor : WORD ;
   DT_4_ToHMI : WORD ;
   DT_4_Floor : WORD ;
   DT_5_ToHMI : WORD ;
   DT_5_Floor : WORD ;
   Humi_1 : REAL ;
   Temp_1 : REAL ;
   Humi_2 : REAL ;
   Temp_2 : REAL ;
   Humi_3 : REAL ;
   Temp_3 : REAL ;
   Humi_4 : REAL ;
   Temp_4 : REAL ;
   Humi_5 : REAL ;
   Temp_5 : REAL ;
   Humi_6 : REAL ;
   Temp_6 : REAL ;
   Humi_7 : REAL ;
   Temp_7 : REAL ;
   Humi_8 : REAL ;
   Temp_8 : REAL ;
   Humi_9 : REAL ;
   Temp_9 : REAL ;
   Humi_10 : REAL ;
   Temp_10 : REAL ;
   Humi_11 : REAL ;
   Temp_11 : REAL ;
   Humi_12 : REAL ;
   Temp_12 : REAL ;
   Humi_13 : REAL ;
   Temp_13 : REAL ;
   Humi_14 : REAL ;
   Temp_14 : REAL ;
   Humi_15 : REAL ;
   Temp_15 : REAL ;
   Humi_16 : REAL ;
   Temp_16 : REAL ;
   Humi_17 : REAL ;
   Temp_17 : REAL ;
   Humi_18 : REAL ;
   Temp_18 : REAL ;
   Humi_19 : REAL ;
   Temp_19 : REAL ;
   Humi_20 : REAL ;
   Temp_20 : REAL ;
   Humi_21 : REAL ;
   Temp_21 : REAL ;
   Humi_22 : REAL ;
   Temp_22 : REAL ;
   Humi_23 : REAL ;
   Temp_23 : REAL ;
   Humi_24 : REAL ;
   Temp_24 : REAL ;
   Humi_25 : REAL ;
   Temp_25 : REAL ;
   Humi_26 : REAL ;
   Temp_26 : REAL ;
   Humi_27 : REAL ;
   Temp_27 : REAL ;
   Humi_28 : REAL ;
   Temp_28 : REAL ;
   Humi_29 : REAL ;
   Temp_29 : REAL ;
   Humi_30 : REAL ;
   Temp_30 : REAL ;
   Humi_31 : REAL ;
   Temp_31 : REAL ;
   Humi_32 : REAL ;
   Temp_32 : REAL ;
   Humi_33 : REAL ;
   Temp_33 : REAL ;
   Humi_34 : REAL ;
   Temp_34 : REAL ;
   Humi_35 : REAL ;
   Temp_35 : REAL ;
   Humi_36 : REAL ;
   Temp_36 : REAL ;
   Humi_37 : REAL ;
   Temp_37 : REAL ;
   Humi_38 : REAL ;
   Temp_38 : REAL ;
   Humi_39 : REAL ;
   Temp_39 : REAL ;
   Humi_40 : REAL ;
   Temp_40 : REAL ;
   Humi_41 : REAL ;
   Temp_41 : REAL ;
   Humi_42 : REAL ;
   Temp_42 : REAL ;
   Humi_43 : REAL ;
   Temp_43 : REAL ;
   Humi_44 : REAL ;
   Temp_44 : REAL ;
   Humi_45 : REAL ;
   Temp_45 : REAL ;
   Humi_46 : REAL ;
   Temp_46 : REAL ;
   Humi_47 : REAL ;
   Temp_47 : REAL ;
   Humi_48 : REAL ;
   Temp_48 : REAL ;
   Humi_49 : REAL ;
   Temp_49 : REAL ;
   Humi_50 : REAL ;
   Temp_50 : REAL ;
   Humi_51 : REAL ;
   Temp_51 : REAL ;
   Humi_52 : REAL ;
   Temp_52 : REAL ;
   Humi_53 : REAL ;
   Temp_53 : REAL ;
   Humi_54 : REAL ;
   Temp_54 : REAL ;
   Humi_55 : REAL ;
   Temp_55 : REAL ;
   Humi_56 : REAL ;
   Temp_56 : REAL ;
   Humi_57 : REAL ;
   Temp_57 : REAL ;
   Humi_58 : REAL ;
   Temp_58 : REAL ;
   Humi_59 : REAL ;
   Temp_59 : REAL ;
   Humi_60 : REAL ;
   Temp_60 : REAL ;
   CO2_1 : REAL ;
   CO2_2 : REAL ;
   CO2_3 : REAL ;
   CO2_4 : REAL ;
   CO2_5 : REAL ;
   CO2_6 : REAL ;
   CO2_7 : REAL ;
   CO2_8 : REAL ;
   CO2_9 : REAL ;
   CO2_10 : REAL ;
   CO2_11 : REAL ;
   CO2_12 : REAL ;
   CO2_13 : REAL ;
   CO2_14 : REAL ;
   CO2_15 : REAL ;
   CO2_16 : REAL ;
   CO2_17 : REAL ;
   CO2_18 : REAL ;
   CO2_19 : REAL ;
   CO2_20 : REAL ;
   SDPF_1_ToHMI : WORD ;
   SDPF_1_PFB : REAL ;
   SDPF_2_ToHMI : WORD ;
   SDPF_2_PFB : REAL ;
   SDPF_3_ToHMI : WORD ;
   SDPF_3_PFB : REAL ;
   SDPF_4_ToHMI : WORD ;
   SDPF_4_PFB : REAL ;
   SDPF_5_ToHMI : WORD ;
   SDPF_5_PFB : REAL ;
   SDPF_6_ToHMI : WORD ;
   SDPF_6_PFB : REAL ;
   SDPF_7_ToHMI : WORD ;
   SDPF_7_PFB : REAL ;
   SDPF_8_ToHMI : WORD ;
   SDPF_8_PFB : REAL ;
   SDPF_9_ToHMI : WORD ;
   SDPF_9_PFB : REAL ;
   SDPF_10_ToHMI : WORD ;
   SDPF_10_PFB : REAL ;
   EPSA_WLE_1_ToHMI : WORD ;
   EPSA_WLE_2_ToHMI : WORD ;
   EPSA_WLE_3_ToHMI : WORD ;
   EPSA_WLE_4_ToHMI : WORD ;
   EPSA_WLE_5_ToHMI : WORD ;
   EPSA_WLE_6_ToHMI : WORD ;
   EPSA_WLE_7_ToHMI : WORD ;
   EPSA_WLE_8_ToHMI : WORD ;
   EPSB_WLE_1_ToHMI : WORD ;
   EPSB_WLE_2_ToHMI : WORD ;
   EPSB_WLE_3_ToHMI : WORD ;
   EPSB_WLE_4_ToHMI : WORD ;
   EPSB_WLE_5_ToHMI : WORD ;
   EPSB_WLE_6_ToHMI : WORD ;
   EPSB_WLE_7_ToHMI : WORD ;
   EPSB_WLE_8_ToHMI : WORD ;
   XFDF_1_TOHMI : WORD ;
   XFDF_2_TOHMI : WORD ;
   XFDF_3_TOHMI : WORD ;
   XFDF_4_TOHMI : WORD ;
   EPS21_TOHMI1 : WORD ;	//A端
   EPS21_TOHMI : ARRAY  [0 .. 15 ] OF INT ;
   EPS11_TOHMI1 : WORD ;
   EPS11_TOHMI : ARRAY  [0 .. 15 ] OF INT ;
   EPS22_TOHMI1 : WORD ;	//B端
   EPS22_TOHMI : ARRAY  [0 .. 15 ] OF INT ;
   EPS12_TOHMI1 : WORD ;
   EPS12_TOHMI : ARRAY  [0 .. 15 ] OF INT ;
   UPS_ToHMI : WORD ;
   UPS_ToHMI1 : ARRAY  [0 .. 11 ] OF INT ;
   systemStatus : ARRAY  [0 .. 5 ] OF WORD ;	//LSQK
   firstUnitStatus : ARRAY  [0 .. 15 ] OF WORD ;
   secondUnitStatus : ARRAY  [0 .. 15 ] OF WORD ;
   thirdUnitStatus : ARRAY  [0 .. 15 ] OF WORD ;
  END_STRUCT ;	
BEGIN
   DTS_A6_ToHMI := W#16#8002;
   DM_A2_ToHMI := W#16#8012;
END_DATA_BLOCK

